# B&R Automation Studio project NAINV104C00R8L515F00 (part 19)

#### Act_Background.st - Do Not Change!!!
```iecst
(** 2022-12-20 **)
ACTION Act_Background:

	pa_tyAlmData[1]	:= tyAlmData;

	IF (bRstErr = TRUE) THEN

		bErr		:= FALSE;
		bWarning	:= FALSE;

		//Reset Warning
		memset(ADR(a_tyWarningCurrList) , 0 , SIZEOF(a_tyWarningCurrList));
		udiWarningMax	:=1;

		memset(ADR(a_tyCurrList) , 0 , SIZEOF(a_tyCurrList));
		memset(ADR(a_sRecoveryList) , 0 , SIZEOF(a_sRecoveryList));
		memset(ADR(a_udiRecoveryList),0,SIZEOF(a_udiRecoveryList));

		udiAlmCntr	:= 0;

		bAlmUpdt	:= FALSE;

	END_IF

	IF (bRstWarning = TRUE) THEN

		IF bErr =FALSE AND bWarning= TRUE THEN
			//Reset Warning
			memset(ADR(a_tyWarningCurrList) , 0 , SIZEOF(a_tyWarningCurrList));
			udiWarningMax	:=1;

			memset(ADR(a_tyCurrList) , 0 , SIZEOF(a_tyCurrList));
			memset(ADR(a_sRecoveryList) , 0 , SIZEOF(a_sRecoveryList));
			memset(ADR(a_udiRecoveryList),0,SIZEOF(a_udiRecoveryList));
			udiAlmCntr	:= 0;
			bWarning := FALSE;
		END_IF

		bAlmUpdt	:= FALSE;

	END_IF

	IF bAlarmLog = TRUE  AND p_bStartupUISettingsLoadDone THEN

		IF (bAlmUpdt = FALSE) OR (eStatus = Error) THEN

			bInfo		:= FALSE;
			bInfoLF		:= FALSE;
			sInfoMsg	:= '';
			iInfoCntr	:= 0;

			FOR udi := 1 TO p_udiCurrMax DO

				IF (pa_tyAlmData[udi].udiRunTime <> a_udiRunTimeOld[udi]) AND pa_tyAlmData[udi].udiCode <> 0
					AND ((pa_tyAlmData[udi].eSeverity = AlmSeverityError ) ) THEN

					a_udiRunTimeOld[udi]	:= pa_tyAlmData[udi].udiRunTime;

					bAlmUpdt	:= TRUE;

					udiAlmCntr	:= udiAlmCntr + 1;
					IF udiAlmCntr > p_udiCurrMax THEN
						udiAlmCntr	:= p_udiCurrMax;
					END_IF

					udiLogCntr	:= udiLogCntr + 1;
					IF udiLogCntr > p_udiCurrMax THEN
						udiLogCntr	:= p_udiCurrMax;
					END_IF

					fLogDTConvert(ADR(sDT) , p_dtCurrDT);
					udiErrorCode := (pa_tyAlmData[udi].udiCode - 10000) + (pa_tyAlmData[udi].udiModuleNum);//*For HMI Text Group*

					//In this case, Program Name/Data Time/
					//Current List
					a_tyCurrList[udiAlmCntr].eSeverity		:= pa_tyAlmData[udi].eSeverity;
					a_tyCurrList[udiAlmCntr].sProgNm		:= pa_tyAlmData[udi].sProgNm;
					a_tyCurrList[udiAlmCntr].sDT			:= sDT;

					//To HMI Text Group
					a_tyCurrList[udiAlmCntr].udiErrorCode	:= udiErrorCode;
					a_tyCurrList[udiAlmCntr].bAlm			:= pa_tyAlmData[udi].bAlm;

					//Recovery List
					a_sRecoveryList[udiAlmCntr]	 			:= pa_tyAlmData[udi].sRcyMsg;
					a_udiRecoveryList[udiAlmCntr]			:= udiErrorCode; //*For HMI Text Group **It will be the same procedure with the above**

					//History List
					memmove(ADR(a_tyHistoryList[2]) , ADR(a_tyHistoryList[1]) , SIZEOF(a_tyHistoryList[1]) * (p_udiHistoryMax - 1));

					a_tyHistoryList[1].sProgNm			:= pa_tyAlmData[udi].sProgNm;
					a_tyHistoryList[1].sDT				:= sDT;
					a_tyHistoryList[1].udiModErrCode	:= pa_tyAlmData[udi].udiCode;
					a_tyHistoryList[1].udiErrorCode		:= udiErrorCode;

					//Log List
					fLogAlmDispMsg(ADR(sAlmMsg) , p_dtCurrDT , pa_tyAlmData[udi].sProgNm , pa_tyAlmData[udi].udiCode , pa_tyAlmData[udi].sAlmMsg); // *For Log files*
					a_sLogList[udiLogCntr]	:= sAlmMsg;
					a_sLogList[udiLogCntr]	:= CONCAT(a_sLogList[udiLogCntr] , '$r$n');

					//Severity
					IF pa_tyAlmData[udi].eSeverity = AlmSeverityError THEN
						bErr		:= TRUE;
					END_IF

					// Alarm warning
				ELSIF (( pa_tyAlmData[udi].eSeverity = AlmSeverityWarning) AND  (pa_tyAlmData[udi].udiCode <> 0 )) THEN

					//Used to compare
					memset(ADR(sWarningCompareMsg) , 0 , SIZEOF(sWarningCompareMsg));

					sWarningCompareMsg	:= CONCAT(sWarningCompareMsg , pa_tyAlmData[udi].sProgNm);
					sWarningCompareMsg	:= CONCAT(sWarningCompareMsg , ' | ');
					sWarningID := UDINT_TO_STRING(pa_tyAlmData[udi].udiCode);
					sWarningCompareMsg	:= CONCAT(sWarningCompareMsg , sWarningID);
					sWarningCompareMsg	:= CONCAT(sWarningCompareMsg , ' | ');
					sWarningCompareMsg	:= CONCAT(sWarningCompareMsg , pa_tyAlmData[udi].sAlmMsg);

					//Checking whether it is recorded in the alarm list
					FOR udi1 := 0 TO  udiWarningMax DO
						WarningListOccur := (memcmp(ADR(sWarningCompareMsg),ADR(a_tyWarningCurrList[udi1].sMsg),SIZEOF(sWarningCompareMsg) )= 0);

						IF WarningListOccur THEN
							EXIT;
						END_IF

					END_FOR

					//IF warning message is no recorded in alarm list
					IF 	WarningListOccur =FALSE THEN

						bAlmUpdt	:= TRUE;
						udiWarningMax := udiWarningMax +1;

						udiAlmCntr	:= udiAlmCntr + 1;

						IF udiAlmCntr > p_udiCurrMax THEN
							udiAlmCntr	:= p_udiCurrMax;
						END_IF

						udiRecorded[udiWarningMax-1]:= udi;

						udiLogCntr	:= udiLogCntr + 1;

						IF udiLogCntr > p_udiCurrMax THEN
							udiLogCntr	:= p_udiCurrMax;
						END_IF

						//Warning List
						a_tyWarningCurrList[udiWarningMax-1].sMsg		:= sWarningCompareMsg;

						fLogDTConvert(ADR(sDT) , p_dtCurrDT);
						udiErrorCode := (pa_tyAlmData[udi].udiCode - 10000) + pa_tyAlmData[udi].udiModuleNum; //*For HMI Text Group*

						//Current List
						a_tyCurrList[udiAlmCntr].eSeverity		:= pa_tyAlmData[udi].eSeverity;
						a_tyCurrList[udiAlmCntr].sProgNm		:= pa_tyAlmData[udi].sProgNm;
						a_tyCurrList[udiAlmCntr].sDT			:= sDT;
						a_tyCurrList[udiAlmCntr].udiModErrCode	:= pa_tyAlmData[udi].udiCode;

						//To HMI Text Group
						a_tyCurrList[udiAlmCntr].udiErrorCode	:= udiErrorCode;
						a_tyCurrList[udiAlmCntr].bWarning		:= pa_tyAlmData[udi].bWarning;

						//Recovery List
						a_sRecoveryList[udiAlmCntr]	 	:= pa_tyAlmData[udi].sRcyMsg;
						a_udiRecoveryList[udiAlmCntr]	:= udiErrorCode;

						//History List
						memmove(ADR(a_tyHistoryList[2]) , ADR(a_tyHistoryList[1]) , SIZEOF(a_tyHistoryList[1]) * (p_udiHistoryMax - 1));

						a_tyHistoryList[1].sProgNm			:= pa_tyAlmData[udi].sProgNm;
						a_tyHistoryList[1].sDT				:= sDT;
						a_tyHistoryList[1].udiModErrCode	:= pa_tyAlmData[udi].udiCode;
						a_tyHistoryList[1].udiErrorCode		:= udiErrorCode;

						//Log List
						//Info Message
						fLogAlmDispMsg(ADR(sWarningMsg) , p_dtCurrDT , pa_tyAlmData[udi].sProgNm , pa_tyAlmData[udi].udiCode , pa_tyAlmData[udi].sAlmMsg);

						a_sLogList[udiLogCntr]	:= sWarningMsg;
						a_sLogList[udiLogCntr]	:= CONCAT(a_sLogList[udiLogCntr] , '$r$n');

						bWarning	:= TRUE;

					END_IF

					// Show Info Message
				ELSIF  ((pa_tyAlmData[udi].udiCode <> 0) AND (pa_tyAlmData[udi].eSeverity = AlmSeverityInfo)) THEN

					iInfoCntr	:= iInfoCntr + 1;

					IF iInfoCntr = 1 THEN
						sInfoMsg	:= pa_tyAlmData[udi].sAlmMsg;

						IF pa_tyAlmData[udi].sProgNm = 'Follower' AND pa_tyAlmData[udi].sAlmMsg <>'' THEN

							bInfoLF	:= TRUE;
							bInfo	:= TRUE;

						ELSE
							bInfoLF	:= FALSE;
							bInfo	:= TRUE;
						END_IF

					ELSIF iInfoCntr = 2 THEN
						sInfoMsg	:= CONCAT(sInfoMsg , '$r$n$r$n');
						sInfoMsg	:= CONCAT(sInfoMsg , pa_tyAlmData[udi].sAlmMsg);

					END_IF

				END_IF

			END_FOR

		ELSE

			p_eAct	:= AlarmActAppendLogWriteHistory;
			IF eStatus = Done AND eStat = AlarmActAppendLogWriteHistory THEN
				p_eAct		:= AlarmActIdle;
				bAlmUpdt	:= FALSE;
				udiLogCntr	:= 0;
			END_IF

		END_IF

	END_IF

END_ACTION
```

#### Act_Alarm.st - Do Not Change!!!
```iecst
(** 2019-03-25 **)
ACTION Act_Alarm:

	//Error
	IF EDGEPOS(eStatus = Error) THEN

		tyAlmData.sProgNm		:= p_sProgNm;
		tyAlmData.udiCode		:= udiStatus;
		tyAlmData.eSeverity		:= AlmSeverityError;
		tyAlmData.udiRunTime	:= tyAlmData.udiRunTime + 1;
		tyAlmData.bAlm			:= TRUE;
		tyAlmData.udiModuleNum  := udiModuleNum;
		g_sAlarmProgNm		:= p_sProgNm;

		//Get Error Message
		IF tyAlmData.udiCode < 10000 OR tyAlmData.udiCode > 10099 THEN
			tyAlmData.sAlmMsg	:= 'Unknown';
			tyAlmData.sRcyMsg	:= 'Unknown';
		ELSE
			tyAlmData.sAlmMsg	:= a_tyAlmText[tyAlmData.udiCode].sAlmText;
			tyAlmData.sRcyMsg	:= a_tyAlmText[tyAlmData.udiCode].sRcyText;
		END_IF

		sStatTxt	:= tyAlmData.sAlmMsg;

	ELSIF bRstErr AND (tyAlmData.udiCode <> 0) THEN

		tyAlmData.udiCode	:= 0;
		tyAlmData.eSeverity	:= AlmSeverityNA;
		tyAlmData.sAlmMsg	:= '';
		tyAlmData.sRcyMsg	:= '';
		tyAlmData.bAlm			:= FALSE;
		sStatTxt	:= a_sStatText[eStat];

	END_IF

END_ACTION
```

#### InputRef.var - Do Not Change!!!
```iecst
(*2022-12-20*)
(**)
(*General*)
VAR
	p_udiCurrMax : REFERENCE TO UDINT;
	p_udiHistoryMax : REFERENCE TO UDINT;
END_VAR
(**)
VAR
	p_eAct : REFERENCE TO eAlarmAction;
	p_udiRstErr : REFERENCE TO UDINT;
END_VAR
(**)
(*Configuration*)
VAR
	p_dtCurrDT : REFERENCE TO DATE_AND_TIME;
	pa_tyAlmData : REFERENCE TO ARRAY[1..c_udiAlarmCurrMax] OF tyAlmDat;
	p_udiFileKeepDay : REFERENCE TO UDINT;
	p_sProgNm : REFERENCE TO STRING[15];
	p_bNtSettingsLoadDone : REFERENCE TO BOOL;
	p_bStartupUISettingsLoadDone : REFERENCE TO BOOL;
END_VAR
```

#### Local.var - Do Not Change!!!
```iecst
(*2022-12-20*)
(**)
(*Local Action, State & Status*)
VAR
	eAct : eAlarmAction := AlarmActIdle;
	eStat : eAlarmAction := AlarmActIdle;
	eStatus : eFBStatus := Idle;
	udiStatus : UDINT := 0;
	sStatTxt : STRING[200] := '';
	a_sStatText : ARRAY[0..50] OF STRING[200] := ['Idling','Creating Directory','Deleting Old Alarm Log File','Reading History File','Writing History File','Appending Alarm Log File','Appending Alarm Log File & Writing History File','Resetting History','Background Start Alarm Log','Background Stop Alarm Log',41('')];
END_VAR
(**)
(*Local Alarm*)
VAR
	tyAlmData : tyAlmDat;
	a_tyAlmText : ARRAY[10000..10099] OF tyAlmTxt := [(sAlmText:='Create User Directory Error',sRcyText:='An Error Occurred While Attempting To Create User Directory. Please Contact Nutek For A Possible Solution'),(sAlmText:='Create Alarm Directory Error',sRcyText:='An Error Occurred While Attempting To Create Alarm Directory. Please Contact Nutek For A Possible Solution'),(sAlmText:='Get Directory Info Error While Deleting Old Log',sRcyText:='An Error Was Encountered While Getting Directory Info. Please Contact Nutek For A Possible Solution.'),(sAlmText:='Directory Read Error While Deleting Old Log',sRcyText:='An Error Was Encountered While Reading Directory. Please Contact Nutek For A Possible Solution.'),(sAlmText:='File Delete Error While Deleting Old Log',sRcyText:='An Error Was Encountered While Trying To Delete File. Please Contact Nutek For A Possible Solution.'),(sAlmText:='File Open Error While Reading Alarm History',sRcyText:='An Error Was Encountered While Trying To Open File. Please Contact Nutek For A Possible Solution.'),(sAlmText:='File Read Error While Reading Alarm History',sRcyText:='An Error Was Encountered While Trying To Read File. Please Contact Nutek For A Possible Solution.'),(sAlmText:='File Close Error While Reading Alarm History',sRcyText:='An Error Was Encountered While Trying To Close File. Please Contact Nutek For A Possible Solution.'),(sAlmText:='File Open Error While Writing Alarm History',sRcyText:='An Error Was Encountered While Trying To Open File. Please Contact Nutek For A Possible Solution.'),(sAlmText:='File Create Error While Writing Alarm History',sRcyText:='An Error Was Encountered While Trying To Create File. Please Contact Nutek For A Possible Solution.'),(sAlmText:='File Write Error While Writing Alarm History',sRcyText:='An Error Was Encountered While Trying To Write File. Please Contact Nutek For A Possible Solution.'),(sAlmText:='File Close Error While Writing Alarm History',sRcyText:='An Error Was Encountered While Trying To Close File. Please Contact Nutek For A Possible Solution.'),(sAlmText:='Directory Does Not Exist While Writing Alarm History',sRcyText:='The Directory Does Not Exist. Please Contact Nutek For A Possible Solution.'),(sAlmText:='File Open Error While Writing Alarm Log',sRcyText:='An Error Was Encountered While Trying To Open File. Please Contact Nutek For A Possible Solution.'),(sAlmText:='File Create Error While Writing Alarm Log',sRcyText:='An Error Was Encountered While Trying To Create File. Please Contact Nutek For A Possible Solution.'),(sAlmText:='Get File Info Error While Writing Alarm Log',sRcyText:='An Error Was Encountered While Getting File Info. Please Contact Nutek For A Possible Solution.'),(sAlmText:='File Write Error While Writing Alarm Log',sRcyText:='An Error Was Encountered While Trying To Write File. Please Contact Nutek For A Possible Solution.'),(sAlmText:='File Close Error While Writing Alarm Log',sRcyText:='An Error Was Encountered While Trying To Close File. Please Contact Nutek For A Possible Solution.'),(sAlmText:='Directory Does Not Exist While Writing Alarm Log',sRcyText:='The Directory Does Not Exist. Please Contact Nutek For A Possible Solution.'),(sAlmText:='File Open Error While Writing Alarm History',sRcyText:='An Error Was Encountered While Trying To Open File. Please Contact Nutek For A Possible Solution.'),(sAlmText:='File Create Error While Writing Alarm History',sRcyText:='An Error Was Encountered While Trying To Create File. Please Contact Nutek For A Possible Solution.'),(sAlmText:='File Write Error While Writing Alarm History',sRcyText:='An Error Was Encountered While Trying To Write File. Please Contact Nutek For A Possible Solution.'),(sAlmText:='File Close Error While Writing Alarm History',sRcyText:='An Error Was Encountered While Trying To Close File. Please Contact Nutek For A Possible Solution.'),(sAlmText:='Directory Does Not Exist While Writing Alarm History',sRcyText:='The Directory Does Not Exist. Please Contact Nutek For A Possible Solution.'),(sAlmText:='File Open Error While Writing Alarm Log',sRcyText:='An Error Was Encountered While Trying To Open File. Please Contact Nutek For A Possible Solution.'),(sAlmText:='File Create Error While Writing Alarm Log',sRcyText:='An Error Was Encountered While Trying To Create File. Please Contact Nutek For A Possible Solution.'),(sAlmText:='Get File Info Error While Writing Alarm Log',sRcyText:='An Error Was Encountered While Getting File Info. Please Contact Nutek For A Possible Solution.'),(sAlmText:='File Write Error While Writing Alarm Log',sRcyText:='An Error Was Encountered While Trying To Write File. Please Contact Nutek For A Possible Solution.'),(sAlmText:='File Close Error While Writing Alarm Log',sRcyText:='An Error Was Encountered While Trying To Close File. Please Contact Nutek For A Possible Solution.'),(sAlmText:='Directory Does Not Exist While Writing Alarm Log',sRcyText:='The Directory Does Not Exist. Please Contact Nutek For A Possible Solution.'),(sAlmText:='File Open Error While Resetting Alarm History',sRcyText:='An Error Was Encountered While Trying To Open File. Please Contact Nutek For A Possible Solution.'),(sAlmText:='File Create Error While Resetting Alarm History',sRcyText:='An Error Was Encountered While Trying To Create File. Please Contact Nutek For A Possible Solution.'),(sAlmText:='File Write Error While Resetting Alarm History',sRcyText:='An Error Was Encountered While Trying To Write File. Please Contact Nutek For A Possible Solution.'),(sAlmText:='File Close Error While Resetting Alarm History',sRcyText:='An Error Was Encountered While Trying To Close File. Please Contact Nutek For A Possible Solution.'),(sAlmText:='Directory Does Not Exist While Resetting Alarm History',sRcyText:='The Directory Does Not Exist. Please Contact Nutek For A Possible Solution.'),65((0))];
END_VAR
(**)
(*Local Output*)
VAR
	bErr : BOOL;
	bWarning : BOOL;
	a_tyCurrList : ARRAY[1..c_udiAlarmCurrMax] OF tyAlarmCurr;
	a_sRecoveryList : ARRAY[1..c_udiAlarmCurrMax] OF STRING[200];
	a_udiRecoveryList : ARRAY[1..c_udiAlarmCurrMax] OF UDINT;
	a_sHistoryList : ARRAY[1..c_udiAlarmHistoryMax] OF STRING[200];
	bInfo : BOOL;
	sInfoMsg : STRING[200];
	bHistoryFileNotFound : BOOL;
	bInfoLF : BOOL := FALSE;
END_VAR
(**)
(*Local Input*)
VAR
	udiRstErr : UDINT := 0;
	dtCurrDT : DATE_AND_TIME;
	a_tyAlmData : ARRAY[1..c_udiAlarmCurrMax] OF tyAlmDat;
	udiFileKeepDay : UDINT := 30;
	sProgNm : STRING[15] := 'Alarm';
	bNtSettingsLoadDone : BOOL := TRUE;
END_VAR
(**)
(*Local*)
VAR
	bRstErr : BOOL;
	udiRstErrOld : UDINT;
	bInitDone : BOOL;
	bInitialDone : BOOL;
	bAlarmLog : BOOL;
	usiStep : USINT;
	udi : UDINT;
	iInfoCntr : INT;
	sAlmMsg : STRING[300];
	udiAlmCntr : UDINT;
	udiAlmRecvryCntr : UDINT;
	udiLogCntr : UDINT;
	udiWriteLogCntr : UDINT;
	a_sLogList : ARRAY[1..c_udiAlarmCurrMax] OF STRING[200];
	bAlmUpdt : BOOL;
	dtCurrDTTemp : DATE_AND_TIME;
	a_udiRunTimeOld : ARRAY[1..c_udiAlarmCurrMax] OF UDINT;
	fbDirCreate1 : fbDirCreate;
	fbDirCreate2 : fbDirCreate;
	fbFileAppend1 : fbFileFullAppend;
	fbFileOldDel1 : fbFileOldDel;
	fbFileRead1 : fbFileFullRead;
	fbFileWrite1 : fbFileFullWrite;
	udi1 : UDINT;
	udi2 : UDINT;
	udiRecorded : ARRAY[1..c_udiAlarmCurrMax] OF UDINT;
	udiRecorded1 : UDINT;
	bRstWarning : BOOL;
	udiWarningMax : UDINT := 1;
	sWarningMsg : STRING[300];
	sWarningID : STRING[80] := '';
	sWarningCompareMsg : STRING[300];
	a_tyWarningCurrList : ARRAY[1..c_udiAlarmCurrMax] OF tyAlarmCurr;
	a_tyHistoryList : ARRAY[1..c_udiAlarmHistoryMax] OF tyHistory;
	WarningListOccur : BOOL := TRUE;
	udiErrorCode : UDINT;
	sDT : STRING[80];
	udiModuleNum : UDINT := 5051;
END_VAR
```

### RstErr.typ - Do Not Change!!!
```iecst
(*2018-12-13*)
(**)
(*Action*)

TYPE
	eRstErrAction :
		(
		RstErrActIdle,
		RstErrActRun,
		RstErrActSetSafetyRlyRst,
		RstErrActRstSafetyRlyRst
		);
END_TYPE
```

### RstErr.var - Change By Project
```iecst
(*2019-03-25*)
(**)
(*Action & State & Status*)
VAR
	p_RstErrStat : UDINT;
	p_RstErrStatus : UDINT;
	p_RstErrStatTxt : UDINT;
END_VAR
(**)
(*Alarm*)
(**)
(*Output*)
VAR
	p_RstErrReset : UDINT;
	p_RstErrSafetyRlyRst : UDINT;
END_VAR
```

### Program Logical/RstErr/RstErr (IEC, version 1.00.0) - 1.00.0 - 

#### Init.st - Change By Project
```iecst
(** 2019-03-25 **)
PROGRAM _INIT

	(* Always Change If Project Change *)

	//Pass Address To Global Address For External Use
	//Action, State & Status
	p_RstErrStat	:= ADR(eStat);
	p_RstErrStatus	:= ADR(eStatus);
	p_RstErrStatTxt	:= ADR(sStatTxt);

	//Alarm

	//Output
	p_RstErrReset			:= ADR(udiRstErr);
	p_RstErrSafetyRlyRst	:= ADR(bSafetyRlyRst);

	(* Always Change If Project Change *)

END_PROGRAM
```

#### Act_InitGlobal.st - Change By Project
```iecst
(** 2019-03-25 **)
ACTION Act_InitGlobal:

	(* Always Change If Project Change *)

	//Pass Data To Link

	//Pass Data To Internal Use
	p_eAct ACCESS p_UIRstErrAct;
	p_bManual ACCESS p_UIUIMnlMod;
	p_bSafetyRlySig ACCESS p_DISafetyRlySig;
	p_bNtSettingsLoadDone ACCESS p_StartupNtSettingsLoadDone;

	(* Always Change If Project Change *)

END_ACTION
```

#### Act_LinkAction.st - Change By Project
```iecst
(** 2019-03-29 **)
ACTION Act_LinkAction:

	IF EDGENEG(p_bManual) THEN
		p_eAct	:= RstErrActIdle;
	END_IF

END_ACTION
```

#### Act_InitLocal.st - Do Not Change!!!
```iecst
(** 2019-03-25 **)
ACTION Act_InitLocal:

	//Input Reference Link To Local Variable
	p_eAct ACCESS ADR(eAct);
	p_bManual ACCESS ADR(bManual);
	p_bSafetyRlySig ACCESS ADR(bSafetyRlySig);
	p_bNtSettingsLoadDone ACCESS ADR(bNtSettingsLoadDone);

END_ACTION
```

#### Act_Initial.st - Do Not Change!!!
```iecst
(** 2019-01-03 **)
ACTION Act_Initial:

	//Initial
	sStatTxt	:= a_sStatText[eStat];

	fbSafetyRlyRstTm(IN := FALSE);

END_ACTION
```

#### Act_Action.st - Do Not Change!!!
```iecst
(** 2019-03-25 **)
ACTION Act_Action:

	//Reset Done
	IF eStatus = Done AND p_eAct = RstErrActIdle THEN
		eStat	:= RstErrActIdle;
	END_IF

	//Set p_eAct
	IF eStatus = Idle THEN
		eStat	:= p_eAct;
	END_IF

END_ACTION
```

#### Act_Main.st - Do Not Change!!!
```iecst
(** 2019-01-18 **)
ACTION Act_Main:

	//Main
	CASE eStat OF

		RstErrActIdle:
			IF eStatus <> Idle THEN	//Reset Data
				//Private
				fbSafetyRlyRstTm(IN := FALSE);

				sStatTxt	:= a_sStatText[eStat];

				IF p_bManual = FALSE THEN
					bSafetyRlyRst	:= FALSE;
				END_IF

			END_IF

			IF EDGENEG(p_bManual) THEN
				bSafetyRlyRst	:= FALSE;
			END_IF

			eStatus	:= Idle;

		RstErrActRun:
			IF eStatus = Idle OR eStatus = Busy THEN

				eStatus	:= Busy;

				sStatTxt	:= a_sStatText[eStat];

				IF bSafetyRlyRst=FALSE THEN
					udiRstErr	:= udiRstErr + 1;
				END_IF

				IF p_bSafetyRlySig = FALSE THEN
					bSafetyRlyRst	:= TRUE;
				END_IF

				IF bSafetyRlyRst = TRUE THEN
					fbSafetyRlyRstTm(IN := TRUE, PT := T#500ms);

					IF fbSafetyRlyRstTm.Q = TRUE THEN
						bSafetyRlyRst	:= FALSE;
						eStatus			:= Done;
					END_IF

				ELSE
					eStatus	:= Done;

				END_IF

			END_IF

		RstErrActSetSafetyRlyRst:
			IF eStatus = Idle OR eStatus = Busy THEN

				sStatTxt	:= a_sStatText[eStat];

				//Reset
				fbSafetyRlyRstTm(IN := FALSE);

				bSafetyRlyRst	:= TRUE;
				eStatus			:= Done;

			END_IF

		RstErrActRstSafetyRlyRst:
			IF eStatus = Idle OR eStatus = Busy THEN

				sStatTxt	:= a_sStatText[eStat];

				//Reset
				fbSafetyRlyRstTm(IN := FALSE);

				bSafetyRlyRst	:= FALSE;
				eStatus			:= Done;

			END_IF

	END_CASE

END_ACTION
```

#### InputRef.var - Do Not Change!!!
```iecst
(*2019-03-25*)
(**)
(*General*)
VAR
	p_eAct : REFERENCE TO eRstErrAction;
END_VAR
(**)
(*Configuration*)
VAR
	p_bManual : REFERENCE TO BOOL;
END_VAR
(**)
(*Input*)
VAR
	p_bSafetyRlySig : REFERENCE TO BOOL;
	p_bNtSettingsLoadDone : REFERENCE TO BOOL;
END_VAR
```

#### Local.var - Do Not Change!!!
```iecst
(*2019-04-30*)
(**)
(*Local Action, State & Status*)
VAR
	eAct : eRstErrAction := RstErrActIdle;
	eStat : eRstErrAction := RstErrActIdle;
	eStatus : eFBStatus := Idle;
	sStatTxt : STRING[200] := '';
	a_sStatText : ARRAY[0..50] OF STRING[200] := ['Idling','Running Reset Error','Turning On Safety Relay Reset','Turning Off Safety Relay Reset',47('')];
END_VAR
(**)
(*Local Alarm*)
(**)
(*Local Output*)
VAR
	udiRstErr : UDINT;
	bSafetyRlyRst : BOOL;
END_VAR
(**)
(*Local Input*)
VAR
	bManual : BOOL := FALSE;
	bSafetyRlySig : BOOL;
	bNtSettingsLoadDone : BOOL := TRUE;
END_VAR
(**)
(*Local*)
VAR
	bInitDone : BOOL;
	bInitialDone : BOOL;
	fbSafetyRlyRstTm : TON;
END_VAR
```

### ProdRcp.typ - Change By Project
```iecst
(*2020-06-08*)
(**)
(*Action*)

TYPE
	eProdRcpAction :
		(
		ProdRcpActIdle,
		ProdRcpActCreateDir,
		ProdRcpActAddEdit,
		ProdRcpActDel,
		ProdRcpActGetInfo,
		ProdRcpActGetList,
		ProdRcpActFilter,
		ProdRcpActLoadRcp,
		ProdRcpActAdd,
		ProdRcpActEdit,
		ProdRcpActReadCurrRcp,
		ProdRcpActWriteCurrRcpParam,
		ProdRcpActSaveList,
		ProdRcpActSort,
		ProdRcpActEndCharFilter
		);
END_TYPE

(**)
(*Data*)

TYPE
	tyProdRcpParam : 	STRUCT
		sRcpNm : STRING[254];
		diWidthInUM : DINT;
		diWidthInUM2 : DINT;
		usiMcMod : USINT;
		sDisplayInfo : STRING[30];
		dtLastModified : DATE_AND_TIME;
		usiFlippedBrd : USINT;
		sMatchCode : STRING[30];
	END_STRUCT;
END_TYPE
```

### ProdRcp.var - Change By Project
```iecst
(*2020-06-08*)
(**)
(*Constant*)
VAR CONSTANT
	c_udiProdRcpMax : UDINT := 2000;
END_VAR
(**)
(*Action & State & Status*)
VAR
	p_ProdRcpStat : UDINT;
	p_ProdRcpStatus : UDINT;
	p_ProdRcpStatTxt : UDINT;
END_VAR
(**)
(*Alarm*)
VAR
	p_ProdRcpAlmData : UDINT;
END_VAR
(**)
(*Output*)
VAR
	p_ProdRcpNmExist : UDINT;
	p_ProdRcpNmNotExist : UDINT;
	p_ProdRcpNmEmpty : UDINT;
	p_ProdRcpListFull : UDINT;
	p_ProdRcpCurrList : UDINT;
	p_ProdRcpFilterList : UDINT;
	p_ProdRcpSortedList : UDINT;
	p_ProdRcpScanList : UDINT;
	p_ProdRcpInfoOut : UDINT;
	p_ProdRcpFileNotFound : UDINT;
	p_ProdRcpCurrRcpAll : UDINT;
END_VAR
(**)
VAR
	p_ProdRcpCurrRcp0 : UDINT;
	p_ProdRcpCurrRcp0Nm : UDINT;
	p_ProdRcpCurrRcp0Width : UDINT;
	p_ProdRcpCurrRcp0McMod : UDINT;
	p_ProdRcpCurrRcp0FlippedBrd : UDINT;
	p_ProdRcpCurrRcp0MatchCode : UDINT;
	p_ProdRcpCurrRcp0DisplayInfo : UDINT;
	p_ProdRcpCurrRcp0LastModified : UDINT;
	p_ProdRcpCurrRcp0Width2 : UDINT;
END_VAR
(**)
VAR
	p_ProdRcpCurrRcp1 : UDINT;
	p_ProdRcpCurrRcp1Nm : UDINT;
	p_ProdRcpCurrRcp1Width : UDINT;
	p_ProdRcpCurrRcp1McMod : UDINT;
	p_ProdRcpCurrRcp1FlippedBrd : UDINT;
	p_ProdRcpCurrRcp1MatchCode : UDINT;
	p_ProdRcpCurrRcp1DisplayInfo : UDINT;
	p_ProdRcpCurrRcp1LastModified : UDINT;
	p_ProdRcpCurrRcp1Width2 : UDINT;
END_VAR
(**)
VAR
	p_ProdRcpCurrRcp2 : UDINT;
	p_ProdRcpCurrRcp2Nm : UDINT;
	p_ProdRcpCurrRcp2Width : UDINT;
	p_ProdRcpCurrRcp2McMod : UDINT;
	p_ProdRcpCurrRcp2FlippedBrd : UDINT;
	p_ProdRcpCurrRcp2MatchCode : UDINT;
	p_ProdRcpCurrRcp2DisplayInfo : UDINT;
	p_ProdRcpCurrRcp2LastModified : UDINT;
	p_ProdRcpCurrRcp2Width2 : UDINT;
END_VAR
(**)
VAR
	p_ProdRcpCurrRcp3 : UDINT;
	p_ProdRcpCurrRcp3Nm : UDINT;
	p_ProdRcpCurrRcp3Width : UDINT;
	p_ProdRcpCurrRcp3McMod : UDINT;
	p_ProdRcpCurrRcp3FlippedBrd : UDINT;
	p_ProdRcpCurrRcp3MatchCode : UDINT;
	p_ProdRcpCurrRcp3DisplayInfo : UDINT;
	p_ProdRcpCurrRcp3LastModified : UDINT;
	p_ProdRcpCurrRcp3Width2 : UDINT;
END_VAR
(**)
VAR
	p_ProdRcpCurrRcp4 : UDINT;
	p_ProdRcpCurrRcp4Nm : UDINT;
	p_ProdRcpCurrRcp4Width : UDINT;
	p_ProdRcpCurrRcp4McMod : UDINT;
	p_ProdRcpCurrRcp4FlippedBrd : UDINT;
	p_ProdRcpCurrRcp4MatchCode : UDINT;
	p_ProdRcpCurrRcp4DisplayInfo : UDINT;
	p_ProdRcpCurrRcp4LastModified : UDINT;
	p_ProdRcpCurrRcp4Width2 : UDINT;
END_VAR
(**)
VAR
	p_ProdRcpCurrRcp5 : UDINT;
	p_ProdRcpCurrRcp5Nm : UDINT;
	p_ProdRcpCurrRcp5Width : UDINT;
	p_ProdRcpCurrRcp5McMod : UDINT;
	p_ProdRcpCurrRcp5FlippedBrd : UDINT;
	p_ProdRcpCurrRcp5MatchCode : UDINT;
	p_ProdRcpCurrRcp5DisplayInfo : UDINT;
	p_ProdRcpCurrRcp5LastModified : UDINT;
	p_ProdRcpCurrRcp5Width2 : UDINT;
END_VAR
```

### Program Logical/ProdRcp/ProdRcp (IEC, version 1.00.0) - 1.00.0 - NtRecipe v5.00.0 , NtFileIO v5.00.0 (2018-12-01)

#### Init.st - Change By Project
```iecst
(** 2019-06-10 **)
PROGRAM _INIT

	(* Always Change If Project Change *)

	//Pass Address To Global Address For External Use
	//Action, State & Status
	p_ProdRcpStat		:= ADR(eStat);
	p_ProdRcpStatus		:= ADR(eStatus);
	p_ProdRcpStatTxt	:= ADR(sStatTxt);

	//Alarm
	p_ProdRcpAlmData	:= ADR(tyAlmData);

	//Output
	p_ProdRcpNmExist				:= ADR(bNmExist);
	p_ProdRcpNmNotExist				:= ADR(bNmNotExist);
	p_ProdRcpNmEmpty				:= ADR(bNmEmpty);
	p_ProdRcpListFull				:= ADR(bListFull);
	p_ProdRcpCurrList				:= ADR(a_tyCurrList);
	p_ProdRcpFilterList				:= ADR(a_tyFilterList);
	p_ProdRcpSortedList				:= ADR(a_tySortList);
	p_ProdRcpScanList				:= ADR(a_tyScanList);
	p_ProdRcpInfoOut				:= ADR(tyInfoOut);
	p_ProdRcpFileNotFound			:= ADR(bFileNotFound);
	p_ProdRcpCurrRcpAll				:= ADR(a_tyCurrRcp);
	p_ProdRcpCurrRcp0				:= ADR(a_tyCurrRcp[0]);
	p_ProdRcpCurrRcp0Nm				:= ADR(a_tyCurrRcp[0].sRcpNm);
	p_ProdRcpCurrRcp0Width			:= ADR(a_tyCurrRcp[0].diWidthInUM);
	p_ProdRcpCurrRcp0McMod			:= ADR(a_tyCurrRcp[0].usiMcMod);
	p_ProdRcpCurrRcp0FlippedBrd		:= ADR(a_tyCurrRcp[0].usiFlippedBrd);
	p_ProdRcpCurrRcp0MatchCode		:= ADR(a_tyCurrRcp[0].sMatchCode);
	p_ProdRcpCurrRcp0DisplayInfo	:= ADR(a_tyCurrRcp[0].sDisplayInfo);
	p_ProdRcpCurrRcp0LastModified	:= ADR(a_tyCurrRcp[0].dtLastModified);
	p_ProdRcpCurrRcp0Width2			:= ADR(a_tyCurrRcp[0].diWidthInUM2);

	p_ProdRcpCurrRcp1				:= ADR(a_tyCurrRcp[1]);
	p_ProdRcpCurrRcp1Nm				:= ADR(a_tyCurrRcp[1].sRcpNm);
	p_ProdRcpCurrRcp1Width			:= ADR(a_tyCurrRcp[1].diWidthInUM);
	p_ProdRcpCurrRcp1McMod			:= ADR(a_tyCurrRcp[1].usiMcMod);
	p_ProdRcpCurrRcp1FlippedBrd		:= ADR(a_tyCurrRcp[1].usiFlippedBrd);
	p_ProdRcpCurrRcp1MatchCode		:= ADR(a_tyCurrRcp[1].sMatchCode);
	p_ProdRcpCurrRcp1DisplayInfo	:= ADR(a_tyCurrRcp[1].sDisplayInfo);
	p_ProdRcpCurrRcp1LastModified	:= ADR(a_tyCurrRcp[1].dtLastModified);
	p_ProdRcpCurrRcp1Width2			:= ADR(a_tyCurrRcp[1].diWidthInUM2);

	p_ProdRcpCurrRcp2				:= ADR(a_tyCurrRcp[2]);
	p_ProdRcpCurrRcp2Nm				:= ADR(a_tyCurrRcp[2].sRcpNm);
	p_ProdRcpCurrRcp2Width			:= ADR(a_tyCurrRcp[2].diWidthInUM);
	p_ProdRcpCurrRcp2McMod			:= ADR(a_tyCurrRcp[2].usiMcMod);
	p_ProdRcpCurrRcp2FlippedBrd		:= ADR(a_tyCurrRcp[2].usiFlippedBrd);
	p_ProdRcpCurrRcp2MatchCode		:= ADR(a_tyCurrRcp[2].sMatchCode);
	p_ProdRcpCurrRcp2DisplayInfo	:= ADR(a_tyCurrRcp[2].sDisplayInfo);
	p_ProdRcpCurrRcp2LastModified	:= ADR(a_tyCurrRcp[2].dtLastModified);
	p_ProdRcpCurrRcp2Width2			:= ADR(a_tyCurrRcp[2].diWidthInUM2);

	p_ProdRcpCurrRcp3				:= ADR(a_tyCurrRcp[3]);
	p_ProdRcpCurrRcp3Nm				:= ADR(a_tyCurrRcp[3].sRcpNm);
	p_ProdRcpCurrRcp3Width			:= ADR(a_tyCurrRcp[3].diWidthInUM);
	p_ProdRcpCurrRcp3McMod			:= ADR(a_tyCurrRcp[3].usiMcMod);
	p_ProdRcpCurrRcp3FlippedBrd		:= ADR(a_tyCurrRcp[3].usiFlippedBrd);
	p_ProdRcpCurrRcp3MatchCode		:= ADR(a_tyCurrRcp[3].sMatchCode);
	p_ProdRcpCurrRcp3DisplayInfo	:= ADR(a_tyCurrRcp[3].sDisplayInfo);
	p_ProdRcpCurrRcp3LastModified	:= ADR(a_tyCurrRcp[3].dtLastModified);
	p_ProdRcpCurrRcp3Width2			:= ADR(a_tyCurrRcp[3].diWidthInUM2);

	p_ProdRcpCurrRcp4				:= ADR(a_tyCurrRcp[4]);
	p_ProdRcpCurrRcp4Nm				:= ADR(a_tyCurrRcp[4].sRcpNm);
	p_ProdRcpCurrRcp4Width			:= ADR(a_tyCurrRcp[4].diWidthInUM);
	p_ProdRcpCurrRcp4McMod			:= ADR(a_tyCurrRcp[4].usiMcMod);
	p_ProdRcpCurrRcp4FlippedBrd		:= ADR(a_tyCurrRcp[4].usiFlippedBrd);
	p_ProdRcpCurrRcp4MatchCode		:= ADR(a_tyCurrRcp[4].sMatchCode);
	p_ProdRcpCurrRcp4DisplayInfo	:= ADR(a_tyCurrRcp[4].sDisplayInfo);
	p_ProdRcpCurrRcp4LastModified	:= ADR(a_tyCurrRcp[4].dtLastModified);
	p_ProdRcpCurrRcp4Width2			:= ADR(a_tyCurrRcp[4].diWidthInUM2);

	p_ProdRcpCurrRcp5				:= ADR(a_tyCurrRcp[5]);
	p_ProdRcpCurrRcp5Nm				:= ADR(a_tyCurrRcp[5].sRcpNm);
	p_ProdRcpCurrRcp5Width			:= ADR(a_tyCurrRcp[5].diWidthInUM);
	p_ProdRcpCurrRcp5McMod			:= ADR(a_tyCurrRcp[5].usiMcMod);
	p_ProdRcpCurrRcp5FlippedBrd		:= ADR(a_tyCurrRcp[5].usiFlippedBrd);
	p_ProdRcpCurrRcp5MatchCode		:= ADR(a_tyCurrRcp[5].sMatchCode);
	p_ProdRcpCurrRcp5DisplayInfo	:= ADR(a_tyCurrRcp[5].sDisplayInfo);
	p_ProdRcpCurrRcp5LastModified	:= ADR(a_tyCurrRcp[5].dtLastModified);
	p_ProdRcpCurrRcp5Width2			:= ADR(a_tyCurrRcp[5].diWidthInUM2);

	(* Always Change If Project Change *)

END_PROGRAM
```

#### Act_InitGlobal.st - Change By Project
```iecst
(** 2020-06-08 **)
ACTION Act_InitGlobal:

	(* Always Change If Project Change *)

	//Pass Data To Link
	p_bLinkStartupRun ACCESS p_StartupRun;
	p_bLinkNtParamLCSManageRcpPrep ACCESS p_NtParamLCSManageRcpPrep;
	p_bLinkMcParamLCSManageRcpEn ACCESS p_McParamLCSManageRcpEn;
	p_eLinkLCSMngRcpProdRcpAct ACCESS p_LCSMngRcpProdRcpAct;
	p_eLinkUIProdRcpAct ACCESS p_UIProdRcpAct;

	//Pass Data To Internal Use
	p_udiRstErr ACCESS p_RstErrReset;
	p_dtCurrDT ACCESS p_TimeCurrDT;
	p_sSearch ACCESS p_UIProdRcpSearch;
	p_sScan ACCESS p_UIProdRcpScan;
	p_tyInfoIn ACCESS p_UIProdRcpInfoIn;
	p_tyCurrRcpWr ACCESS p_UIProdRcpCurrRcpWr;
	p_sListFileName ACCESS p_NtParamProdRcpListFileNm;
	p_sSingleFileName ACCESS p_NtParamProdRcpSingleFileNm;
	p_sProgNm ACCESS p_NtParamProdRcpProgNm;
	p_bNtSettingsLoadDone ACCESS p_StartupNtSettingsLoadDone;

	p_bWidth2Prep ACCESS p_NtParamLFWidth2Prep;
	(* Always Change If Project Change *)

END_ACTION
```

#### InputRef_Link.var - Change By Project
```iecst
(*2019-04-24*)
(**)
VAR
	rWidthInMM : REAL;
	rWidthInMM2 : REAL;
	sWidthInMM : STRING[30];
	sWidthInMM2 : STRING[30];
	p_bLinkStartupRun : REFERENCE TO BOOL;
	p_bLinkNtParamLCSManageRcpPrep : REFERENCE TO BOOL;
	p_bLinkMcParamLCSManageRcpEn : REFERENCE TO BOOL;
	p_eLinkLCSMngRcpProdRcpAct : REFERENCE TO eProdRcpAction;
	p_eLinkUIProdRcpAct : REFERENCE TO eProdRcpAction;
	udi : UDINT;
	udiSortCurrenTotalCntr : UDINT;
	iSortCurrentOuterCntr : INT;
	iTotalRcp : INT;
	iSortCurrentInnerCntr : INT;
	sDebug : STRING[300];
	tyTempRecipe : tyProdRcpParam;
END_VAR
```

#### Act_LinkAction.st - Change By Project
```iecst
(** 2019-05-20 **)
ACTION Act_LinkAction:

	IF p_bLinkStartupRun = TRUE THEN
		p_eAct ACCESS p_StartupProdRcpAct;
	ELSE
		IF eStatus = Idle THEN
			IF p_bLinkNtParamLCSManageRcpPrep AND p_bLinkMcParamLCSManageRcpEn THEN
				IF p_eLinkLCSMngRcpProdRcpAct <> ProdRcpActIdle THEN
					p_eAct ACCESS p_LCSMngRcpProdRcpAct;
					p_tyInfoIn ACCESS p_LCSMngRcpProdRcpInfoIn;
				ELSIF p_eLinkUIProdRcpAct <> ProdRcpActIdle THEN
					p_eAct ACCESS p_UIProdRcpAct;
					p_tyInfoIn ACCESS p_UIProdRcpInfoIn;

					p_tyInfoIn.dtLastModified	:= p_dtCurrDT;
				END_IF
			ELSE
				p_eAct ACCESS p_UIProdRcpAct;
				p_tyInfoIn ACCESS p_UIProdRcpInfoIn;

				p_tyInfoIn.dtLastModified	:= p_dtCurrDT;
			END_IF
		END_IF
	END_IF

END_ACTION
```

#### Act_Link.st - Change By Project
```iecst
(** 2019-04-30 **)
ACTION Act_Link:

	IF (p_eAct = ProdRcpActAddEdit) OR (p_eAct = ProdRcpActAdd) OR (p_eAct = ProdRcpActEdit) THEN

		rWidthInMM				:= DINT_TO_REAL(p_tyInfoIn.diWidthInUM);
		rWidthInMM2				:= DINT_TO_REAL(p_tyInfoIn.diWidthInUM2);
		rWidthInMM				:= rWidthInMM / 1000;
		rWidthInMM2				:= rWidthInMM2 / 1000;
		sWidthInMM				:= REAL_TO_STRING(rWidthInMM);
		sWidthInMM2				:= REAL_TO_STRING(rWidthInMM2);

		IF p_bWidth2Prep THEN
			p_tyInfoIn.sDisplayInfo	:= sWidthInMM;
			p_tyInfoIn.sDisplayInfo	:= CONCAT(p_tyInfoIn.sDisplayInfo , ' | ');
			p_tyInfoIn.sDisplayInfo	:= CONCAT(p_tyInfoIn.sDisplayInfo , sWidthInMM2);
			p_tyInfoIn.sDisplayInfo	:= CONCAT(p_tyInfoIn.sDisplayInfo , ' mm');
		ELSE
			p_tyInfoIn.sDisplayInfo	:= sWidthInMM;
			p_tyInfoIn.sDisplayInfo	:= CONCAT(p_tyInfoIn.sDisplayInfo , ' mm');
		END_IF
	END_IF

END_ACTION
```

#### Cyclic.st - Do Not Change!!!
```iecst
(** 2019-03-29 **)
PROGRAM _CYCLIC

	IF bInitDone = FALSE THEN
		bInitDone	:= TRUE;

		Act_InitLocal;
		Act_InitGlobal;

	ELSIF bInitialDone = FALSE THEN
		IF p_bNtSettingsLoadDone = TRUE THEN
			bInitialDone	:= TRUE;

			Act_Initial;
		END_IF

	ELSE

		Act_RstErr;
		Act_LinkAction;
		Act_Action;
		Act_Link;
		Act_Main;
		Act_Alarm;

	END_IF

END_PROGRAM
```

#### Act_InitLocal.st - Do Not Change!!!
```iecst
(** 2020-06-08 **)
ACTION Act_InitLocal:

	//Input Reference Link To Local Variable
	p_eAct ACCESS ADR(eAct);
	p_udiMax ACCESS ADR(c_udiProdRcpMax);
	p_udiRstErr ACCESS ADR(udiRstErr);
	p_dtCurrDT ACCESS ADR(dtCurrDT);
	p_sSearch ACCESS ADR(sSearch);
	p_sScan ACCESS ADR(sScan);
	p_tyInfoIn ACCESS ADR(tyInfoIn);
	p_tyCurrRcpWr ACCESS ADR(tyCurrRcpWr);
	p_sListFileName ACCESS ADR(sListFileName);
	p_sSingleFileName ACCESS ADR(sSingleFileName);
	p_sProgNm ACCESS ADR(sProgNm);
	p_bNtSettingsLoadDone ACCESS ADR(bNtSettingsLoadDone);
	p_bWidth2Prep ACCESS ADR(bWidth2Prep);

END_ACTION
```

#### Act_Initial.st - Do Not Change!!!
```iecst
(** 2019-06-10 **)
ACTION Act_Initial:

	//Initial
	sStatTxt	:= a_sStatText[eStat];

	fbDirCreate1.sDevice	:= 'F';
	fbDirCreate1.sDirName	:= 'User';
	fbDirCreate1(bEn := FALSE);

	fbDirCreate2.sDevice	:= 'User';
	fbDirCreate2.sDirName	:= 'ProductRecipe';
	fbDirCreate2(bEn := FALSE);

	fbFileReadList.sDevice		:= 'ProdRcp';
	fbFileReadList.sFile		:= p_sListFileName;
	fbFileReadList.udiOffset	:= 0;
	fbFileReadList.p_Dest		:= ADR(a_tyCurrList);
	fbFileReadList.udiLen		:= SIZEOF(a_tyCurrList);
	fbFileReadList(bEn := FALSE);

	fbFileWriteList.sDevice		:= 'ProdRcp';
	fbFileWriteList.sFile		:= p_sListFileName;
	fbFileWriteList.udiOffset	:= 0;
	fbFileWriteList.p_Src		:= ADR(a_tyListTemp);
	fbFileWriteList.udiLen		:= SIZEOF(a_tyListTemp);
	fbFileWriteList.udiOption	:= 0;
	fbFileWriteList(bEn := FALSE);

	fbFileReadSingle.sDevice	:= 'ProdRcp';
	fbFileReadSingle.sFile		:= p_sSingleFileName;
	fbFileReadSingle.udiOffset	:= 0;
	fbFileReadSingle.p_Dest		:= ADR(a_tyCurrRcp[0]);
	fbFileReadSingle.udiLen		:= SIZEOF(a_tyCurrRcp[0]);
	fbFileReadSingle(bEn := FALSE);

	fbFileLoadSingle.sDevice	:= 'ProdRcp';
	fbFileLoadSingle.sFile		:= p_sSingleFileName;
	fbFileLoadSingle.udiOffset	:= 0;
	fbFileLoadSingle.p_Src		:= ADR(a_tyCurrRcp[0]);
	fbFileLoadSingle.udiLen		:= SIZEOF(a_tyCurrRcp[0]);
	fbFileLoadSingle.udiOption	:= 0;
	fbFileLoadSingle(bEn := FALSE);

	fbFileWriteSingle.sDevice	:= 'ProdRcp';
	fbFileWriteSingle.sFile		:= p_sSingleFileName;
	fbFileWriteSingle.udiOffset	:= 0;
	fbFileWriteSingle.p_Src		:= ADR(p_tyCurrRcpWr);
	fbFileWriteSingle.udiLen	:= SIZEOF(p_tyCurrRcpWr);
	fbFileWriteSingle.udiOption	:= 0;
	fbFileWriteSingle(bEn := FALSE);

END_ACTION
```

#### Act_Action.st - Do Not Change!!!
```iecst
(** 2019-03-25 **)
ACTION Act_Action:

	//Reset Error
	IF (eStatus = Error) AND bRstErr THEN
		p_eAct	:= ProdRcpActIdle;
		eStat	:= ProdRcpActIdle;
	END_IF

	//Reset Done
	IF eStatus = Done AND p_eAct = ProdRcpActIdle THEN
		eStat	:= ProdRcpActIdle;
	END_IF

	//Set p_eAct
	IF eStatus = Idle THEN
		eStat	:= p_eAct;
	END_IF

END_ACTION
```

#### Act_Main.st - Do Not Change!!!
```iecst
(** 2023-02-13 **)
ACTION Act_Main:

	//Main
	CASE eStat OF

		ProdRcpActIdle:
			IF eStatus <> Idle THEN	//Reset Data
				//Private
				fbDirCreate1(bEn := FALSE);
				fbDirCreate2(bEn := FALSE);
				fbFileReadList(bEn := FALSE);
				fbFileWriteList(bEn := FALSE);
				fbFileReadSingle(bEn := FALSE);
				fbFileWriteSingle(bEn := FALSE);
				fbFileLoadSingle(bEn := FALSE);
				usiStep				:= 0;
				udiAddStatus		:= 0;

				bNmExist		:= FALSE;
				bNmNotExist		:= FALSE;
				bNmEmpty		:= FALSE;
				bListFull		:= FALSE;
				bFileNotFound	:= FALSE;
				iTotalRcp 		:= 0;

				memset(ADR(tyTempRecipe), 0 , SIZEOF(tyTempRecipe));

				sStatTxt	:= a_sStatText[eStat];

			END_IF

			eStatus	:= Idle;

		ProdRcpActCreateDir:
			IF eStatus = Idle OR eStatus = Busy THEN

				eStatus	:= Busy;

				sStatTxt	:= a_sStatText[eStat];

				CASE usiStep OF
					0:
						fbDirCreate1(bEn := TRUE);
						IF fbDirCreate1.udiStatus = 0 THEN
							usiStep	:= 1;
						ELSIF fbDirCreate1.udiStatus < 65534 THEN
							eStatus		:= Error;

							IF fbDirCreate1.udiStatus = 1908 THEN
								udiStatus	:= 10000;	//Create User Directory Error
							ELSE
								udiStatus	:= fbDirCreate1.udiStatus;
							END_IF
						END_IF

					1:
						fbDirCreate2(bEn := TRUE);
						IF fbDirCreate2.udiStatus = 0 THEN
							eStatus	:= Done;
						ELSIF fbDirCreate2.udiStatus < 65534 THEN
							eStatus		:= Error;

							IF fbDirCreate2.udiStatus = 1908 THEN
								udiStatus	:= 10001;	//Create Product Recipe Directory Error
							ELSE
								udiStatus	:= fbDirCreate2.udiStatus;
							END_IF
						END_IF

				END_CASE

			END_IF

		ProdRcpActAddEdit:
			IF eStatus = Idle OR eStatus = Busy THEN

				eStatus	:= Busy;

				sStatTxt	:= a_sStatText[eStat];

				CASE usiStep OF
					0:	//Edit Recipe
						udiAddStatus	:= fRecipeAddEdit(ADR(p_tyInfoIn) , ADR(a_tyListTemp) , SIZEOF(a_tyListTemp[1]) , ADR(a_tyListTemp[1].sRcpNm) , SIZEOF(a_tyListTemp[1].sRcpNm) , p_udiMax);

						IF udiAddStatus = 1600 THEN	//Recipe Name Empty
							bNmEmpty	:= TRUE;
							eStatus		:= Done;

						ELSIF udiAddStatus = 1601 THEN	//Recipe Full
							bListFull	:= TRUE;
							eStatus		:= Done;

						ELSIF udiAddStatus = 0 THEN	//OK
							usiStep	:= 1;

						END_IF

					1:	//Write Into File
						fbFileWriteList(bEn := TRUE);

						IF fbFileWriteList.udiStatus = 0 THEN
							a_tyCurrList	:= a_tyListTemp;

							eStatus := Done;

						ELSIF fbFileWriteList.udiStatus < 65534 THEN
							a_tyListTemp	:= a_tyCurrList;
							eStatus			:= Error;

							IF fbFileWriteList.udiStatus = 1900 THEN
								udiStatus	:= 10002;	//File Open Error While Adding & Editing
							ELSIF fbFileWriteList.udiStatus = 1901 THEN
								udiStatus	:= 10003;	//File Create Error While Adding & Editing
							ELSIF fbFileWriteList.udiStatus = 1903 THEN
								udiStatus	:= 10004;	//File Write Error While Adding & Editing
							ELSIF fbFileWriteList.udiStatus = 1904 THEN
								udiStatus	:= 10005;	//File Close Error While Adding & Editing
							ELSIF fbFileWriteList.udiStatus = 1914 THEN
								udiStatus	:= 10013;	//Directory Does Not Exist While Adding & Editing
							ELSE
								udiStatus	:= fbFileWriteList.udiStatus;
							END_IF
						END_IF

				END_CASE

			END_IF

		ProdRcpActDel:
			IF eStatus = Idle OR eStatus = Busy THEN

				eStatus	:= Busy;

				sStatTxt	:= a_sStatText[eStat];

				CASE usiStep OF
					0:	//Edit User
						udiAddStatus	:= fRecipeDelete(ADR(p_tyInfoIn) , ADR(a_tyListTemp) , SIZEOF(a_tyListTemp[1]) , ADR(a_tyListTemp[1].sRcpNm) , SIZEOF(a_tyListTemp[1].sRcpNm) , p_udiMax);

						IF udiAddStatus = 1600 THEN	//Recipe Name Empty
							bNmEmpty	:= TRUE;
							eStatus		:= Done;

						ELSIF udiAddStatus = 1603 THEN	//Recipe Not Exist
							bNmNotExist	:= TRUE;
							eStatus		:= Done;

						ELSIF udiAddStatus = 0 THEN	//OK
							usiStep	:= 1;

						END_IF

					1:	//Write Into File
						fbFileWriteList(bEn := TRUE);

						IF fbFileWriteList.udiStatus = 0 THEN
							a_tyCurrList	:= a_tyListTemp;
							eStatus := Done;

						ELSIF fbFileWriteList.udiStatus < 65534 THEN
							a_tyListTemp	:= a_tyCurrList;
							eStatus			:= Error;

							IF fbFileWriteList.udiStatus = 1900 THEN
								udiStatus	:= 10006;	//File Open Error While Deleting
							ELSIF fbFileWriteList.udiStatus = 1901 THEN
								udiStatus	:= 10007;	//File Create Error While Deleting
							ELSIF fbFileWriteList.udiStatus = 1903 THEN
								udiStatus	:= 10008;	//File Write Error While Deleting
							ELSIF fbFileWriteList.udiStatus = 1904 THEN
								udiStatus	:= 10009;	//File Close Error While Deleting
							ELSIF fbFileWriteList.udiStatus = 1914 THEN
								udiStatus	:= 10014;	//Directory Does Not Exist While Deleting
							ELSE
								udiStatus	:= fbFileWriteList.udiStatus;
							END_IF

						END_IF

				END_CASE

			END_IF

		ProdRcpActGetInfo:
			IF eStatus = Idle OR eStatus = Busy THEN

				sStatTxt	:= a_sStatText[eStat];

				IF p_tyInfoIn.sRcpNm = '' THEN
					bNmEmpty	:= TRUE;
					bNmNotExist	:= TRUE;
				ELSE
					bNmNotExist	:= (fRecipeGetInfo(p_tyInfoIn.sRcpNm , ADR(tyInfoOut) , ADR(a_tyCurrList) , SIZEOF(a_tyCurrList[1]) , ADR(a_tyCurrList[1].sRcpNm) , SIZEOF(a_tyCurrList[1].sRcpNm) , p_udiMax)) = 0;
				END_IF

				eStatus	:= Done;

			END_IF

		ProdRcpActGetList:
			IF eStatus = Idle OR eStatus = Busy THEN

				eStatus	:= Busy;

				sStatTxt	:= a_sStatText[eStat];

				fbFileReadList(bEn := TRUE);

				IF fbFileReadList.udiStatus = 0 THEN
					a_tyListTemp	:= a_tyCurrList;
					eStatus			:= Done;

				ELSIF fbFileReadList.udiStatus < 65534 THEN
					eStatus		:= Error;

					IF fbFileReadList.udiStatus = 1900 THEN
						udiStatus	:= 10010;	//File Open Error While Getting List
					ELSIF fbFileReadList.udiStatus = 1902 THEN
						udiStatus	:= 10011;	//File Read Error While Getting List
					ELSIF fbFileReadList.udiStatus = 1904 THEN
						udiStatus	:= 10012;	//File Close Error While Getting List
					ELSIF fbFileReadList.udiStatus = 1915 THEN
						eStatus			:= Done;
						bFileNotFound	:= TRUE;
					ELSE
						udiStatus	:= fbFileReadList.udiStatus;
					END_IF

				END_IF

			END_IF

		ProdRcpActFilter:

			IF eStatus = Idle OR eStatus = Busy THEN

				eStatus := Busy;

				sStatTxt	:= a_sStatText[eStat];

				CASE usiStep OF
					0:
						fRecipeFilter(p_sSearch , ADR(a_tyFilterList) , ADR(a_tyCurrList) , SIZEOF(a_tyCurrList[1]) , ADR(a_tyCurrList[1].sRcpNm) ,
						SIZEOF(a_tyCurrList[1].sRcpNm) , p_udiMax, 0, 499, iFilterCtr);
						usiStep := 1;
					1:
						fRecipeFilter(p_sSearch , ADR(a_tyFilterList) , ADR(a_tyCurrList) , SIZEOF(a_tyCurrList[1]) , ADR(a_tyCurrList[1].sRcpNm) ,
						SIZEOF(a_tyCurrList[1].sRcpNm) , p_udiMax, 500, 999, iFilterCtr);
						usiStep := 2;
					2:
						fRecipeFilter(p_sSearch , ADR(a_tyFilterList) , ADR(a_tyCurrList) , SIZEOF(a_tyCurrList[1]) , ADR(a_tyCurrList[1].sRcpNm) ,
						SIZEOF(a_tyCurrList[1].sRcpNm) , p_udiMax, 1000, 1499, iFilterCtr);
						usiStep := 3;
					3:
						fRecipeFilter(p_sSearch , ADR(a_tyFilterList) , ADR(a_tyCurrList) , SIZEOF(a_tyCurrList[1]) , ADR(a_tyCurrList[1].sRcpNm) ,
						SIZEOF(a_tyCurrList[1].sRcpNm) , p_udiMax, 1500, 1999, iFilterCtr);
						eStatus := Done;

				END_CASE

			END_IF

		ProdRcpActLoadRcp:
			IF eStatus = Idle OR eStatus = Busy THEN

				sStatTxt	:= a_sStatText[eStat];

				CASE usiStep OF
					0:	//Get Current Recipe
						IF p_tyInfoIn.sRcpNm = '' THEN
							bNmEmpty	:= TRUE;
							bNmNotExist	:= TRUE;

							eStatus	:= Done;
						ELSE
							bNmNotExist	:= (fRecipeGetInfo(p_tyInfoIn.sRcpNm , ADR(a_tyCurrRcp[0]) , ADR(a_tyCurrList) , SIZEOF(a_tyCurrList[1]) , ADR(a_tyCurrList[1].sRcpNm) , SIZEOF(a_tyCurrList[1].sRcpNm) , p_udiMax)) = 0;

							IF bNmNotExist = TRUE THEN
								eStatus	:= Done;
							ELSE
								usiStep	:= 1;
							END_IF

						END_IF

					1:	//Write Into File
						fbFileLoadSingle(bEn := TRUE);

						IF fbFileLoadSingle.udiStatus = 0 THEN
							eStatus			:= Done;
						ELSIF fbFileLoadSingle.udiStatus < 65534 THEN
							eStatus			:= Error;

							IF fbFileLoadSingle.udiStatus = 1900 THEN
								udiStatus	:= 10025;	//File Open Error While Loading Current Recipe
							ELSIF fbFileLoadSingle.udiStatus = 1901 THEN
								udiStatus	:= 10026;	//File Create Error While Loading Current Recipe
							ELSIF fbFileLoadSingle.udiStatus = 1903 THEN
								udiStatus	:= 10027;	//File Write Error While Loading Current Recipe
							ELSIF fbFileLoadSingle.udiStatus = 1904 THEN
								udiStatus	:= 10028;	//File Close Error While Loading Current Recipe
							ELSIF fbFileLoadSingle.udiStatus = 1914 THEN
								udiStatus	:= 10029;	//Directory Does Not Exist While Loading Current Recipe
							ELSE
								udiStatus	:= fbFileLoadSingle.udiStatus;
							END_IF
						END_IF

				END_CASE

			END_IF

		ProdRcpActAdd:
			IF eStatus = Idle OR eStatus = Busy THEN

				eStatus	:= Busy;

				sStatTxt	:= a_sStatText[eStat];

				CASE usiStep OF
					0:	//Edit Recipe
						udiAddStatus	:= fRecipeAdd(ADR(p_tyInfoIn) , ADR(a_tyListTemp) , SIZEOF(a_tyListTemp[1]) , ADR(a_tyListTemp[1].sRcpNm) , SIZEOF(a_tyListTemp[1].sRcpNm) , p_udiMax);

						IF udiAddStatus = 1600 THEN	//Recipe Name Empty
							bNmEmpty	:= TRUE;
							eStatus		:= Done;

						ELSIF udiAddStatus = 1601 THEN	//Recipe Full
							bListFull	:= TRUE;
							eStatus		:= Done;

						ELSIF udiAddStatus = 1602 THEN	//Recipe Name Exist
							bNmExist	:= TRUE;
							eStatus		:= Done;

						ELSIF udiAddStatus = 0 THEN	//OK
							usiStep	:= 1;

						END_IF

					1:	//Write Into File
						fbFileWriteList(bEn := TRUE);

						IF fbFileWriteList.udiStatus = 0 THEN
							a_tyCurrList	:= a_tyListTemp;
							eStatus			:= Done;

						ELSIF fbFileWriteList.udiStatus < 65534 THEN
							a_tyListTemp	:= a_tyCurrList;
							eStatus			:= Error;

							IF fbFileWriteList.udiStatus = 1900 THEN
								udiStatus	:= 10015;	//File Open Error While Adding
							ELSIF fbFileWriteList.udiStatus = 1901 THEN
								udiStatus	:= 10016;	//File Create Error While Adding
							ELSIF fbFileWriteList.udiStatus = 1903 THEN
								udiStatus	:= 10017;	//File Write Error While Adding
							ELSIF fbFileWriteList.udiStatus = 1904 THEN
								udiStatus	:= 10018;	//File Close Error While Adding
							ELSIF fbFileWriteList.udiStatus = 1914 THEN
								udiStatus	:= 10019;	//Directory Does Not Exist While Adding
							ELSE
								udiStatus	:= fbFileWriteList.udiStatus;
							END_IF
						END_IF
				END_CASE

			END_IF

		ProdRcpActEdit:
			IF eStatus = Idle OR eStatus = Busy THEN

				eStatus	:= Busy;

				sStatTxt	:= a_sStatText[eStat];

				CASE usiStep OF
					0:	//Edit Recipe
						udiAddStatus	:= fRecipeEdit(ADR(p_tyInfoIn) , ADR(a_tyListTemp) , SIZEOF(a_tyListTemp[1]) , ADR(a_tyListTemp[1].sRcpNm) , SIZEOF(a_tyListTemp[1].sRcpNm) , p_udiMax);

						IF udiAddStatus = 1600 THEN	//Recipe Name Empty
							bNmEmpty	:= TRUE;
							eStatus		:= Done;

						ELSIF udiAddStatus = 1603 THEN	//Recipe Not Exist
							bNmNotExist	:= TRUE;
							eStatus		:= Done;

						ELSIF udiAddStatus = 0 THEN	//OK
							usiStep	:= 1;

						END_IF

					1:	//Write Into File
						fbFileWriteList(bEn := TRUE);

						IF fbFileWriteList.udiStatus = 0 THEN
							a_tyCurrList	:= a_tyListTemp;
							eStatus			:= Done;

						ELSIF fbFileWriteList.udiStatus < 65534 THEN
							a_tyListTemp	:= a_tyCurrList;
							eStatus			:= Error;

							IF fbFileWriteList.udiStatus = 1900 THEN
								udiStatus	:= 10020;	//File Open Error While Adding & Editing
							ELSIF fbFileWriteList.udiStatus = 1901 THEN
								udiStatus	:= 10021;	//File Create Error While Adding & Editing
							ELSIF fbFileWriteList.udiStatus = 1903 THEN
								udiStatus	:= 10022;	//File Write Error While Adding & Editing
							ELSIF fbFileWriteList.udiStatus = 1904 THEN
								udiStatus	:= 10023;	//File Close Error While Adding & Editing
							ELSIF fbFileWriteList.udiStatus = 1914 THEN
								udiStatus	:= 10024;	//Directory Does Not Exist While Adding & Editing
							ELSE
								udiStatus	:= fbFileWriteList.udiStatus;
							END_IF
						END_IF

				END_CASE

			END_IF

		ProdRcpActReadCurrRcp:
			IF eStatus = Idle OR eStatus = Busy THEN

				eStatus	:= Busy;

				sStatTxt	:= a_sStatText[eStat];

				fbFileReadSingle(bEn := TRUE);
				IF fbFileReadSingle.udiStatus = 0 THEN
					eStatus			:= Done;

				ELSIF fbFileReadSingle.udiStatus < 65534 THEN
					eStatus		:= Error;

					IF fbFileReadSingle.udiStatus = 1900 THEN
						udiStatus	:= 10030;	//File Open Error While Reading Current Recipe
					ELSIF fbFileReadSingle.udiStatus = 1902 THEN
						udiStatus	:= 10031;	//File Read Error While Reading Current Recipe
					ELSIF fbFileReadSingle.udiStatus = 1904 THEN
						udiStatus	:= 10032;	//File Close Error While Reading Current Recipe
					ELSIF fbFileReadSingle.udiStatus = 1915 THEN
						eStatus			:= Done;
						bFileNotFound	:= TRUE;
					ELSE
						udiStatus	:= fbFileReadSingle.udiStatus;
					END_IF
				END_IF

			END_IF

		ProdRcpActWriteCurrRcpParam:
			IF eStatus = Idle OR eStatus = Busy THEN

				sStatTxt	:= a_sStatText[eStat];

				fbFileWriteSingle(bEn := TRUE);

				IF fbFileWriteSingle.udiStatus = 0 THEN
					a_tyCurrRcp[0]	:= p_tyCurrRcpWr;
					eStatus			:= Done;
				ELSIF fbFileWriteSingle.udiStatus < 65534 THEN
					eStatus			:= Error;

					IF fbFileWriteSingle.udiStatus = 1900 THEN
						udiStatus	:= 10033;	//File Open Error While Writing Current Recipe Parameter
					ELSIF fbFileWriteSingle.udiStatus = 1901 THEN
						udiStatus	:= 10034;	//File Create Error While Writing Current Recipe Parameter
					ELSIF fbFileWriteSingle.udiStatus = 1903 THEN
						udiStatus	:= 10035;	//File Write Error While Writing Current Recipe Parameter
					ELSIF fbFileWriteSingle.udiStatus = 1904 THEN
						udiStatus	:= 10036;	//File Close Error While Writing Current Recipe Parameter
					ELSIF fbFileWriteSingle.udiStatus = 1914 THEN
						udiStatus	:= 10037;	//Directory Does Not Exist Writing Current Recipe Parameter
					ELSE
						udiStatus	:= fbFileWriteSingle.udiStatus;
					END_IF
				END_IF

			END_IF

		ProdRcpActSaveList:
			IF eStatus = Idle OR eStatus = Busy THEN

				eStatus	:= Busy;

				sStatTxt	:= a_sStatText[eStat];

				CASE usiStep OF

					0:
						a_tyListTemp	:= a_tyCurrList;

						fbFileWriteList(bEn := TRUE);

						IF fbFileWriteList.udiStatus = 0 THEN
							eStatus			:= Done;

						ELSIF fbFileWriteList.udiStatus < 65534 THEN
							eStatus			:= Error;

							IF fbFileWriteList.udiStatus = 1900 THEN
								udiStatus	:= 10038;	//File Open Error While Saving List
							ELSIF fbFileWriteList.udiStatus = 1901 THEN
								udiStatus	:= 10039;	//File Create Error While Saving List
							ELSIF fbFileWriteList.udiStatus = 1903 THEN
								udiStatus	:= 10040;	//File Write Error While Saving List
							ELSIF fbFileWriteList.udiStatus = 1904 THEN
								udiStatus	:= 10041;	//File Close Error While Saving List
							ELSIF fbFileWriteList.udiStatus = 1914 THEN
								udiStatus	:= 10042;	//Directory Does Not Exist While Saving List
							ELSE
								udiStatus	:= fbFileWriteList.udiStatus;
							END_IF
						END_IF

				END_CASE

			END_IF

		ProdRcpActSort:
			IF eStatus = Idle OR eStatus = Busy THEN

				sStatTxt	:= a_sStatText[eStat];

				CASE usiStep OF

					0:

						FOR udi := 1 TO c_udiProdRcpMax DO
							IF p_sSearch <> '' THEN
								IF a_tyFilterList[udi].sRcpNm = '' THEN
									usiStep := 1;
									EXIT;
								ELSIF udi = c_udiProdRcpMax THEN
									iTotalRcp := UDINT_TO_INT(c_udiProdRcpMax);
									usiStep := 1;
									EXIT;
								ELSE
									iTotalRcp := iTotalRcp +1;
								END_IF
							ELSE
								IF a_tyCurrList[udi].sRcpNm = '' THEN
									usiStep := 1;
									EXIT;
								ELSIF udi = c_udiProdRcpMax THEN
									iTotalRcp := UDINT_TO_INT(c_udiProdRcpMax);
									usiStep := 1;
									EXIT;
								ELSE
									iTotalRcp := iTotalRcp +1;
								END_IF
							END_IF
						END_FOR

					1:
						IF p_sSearch <> '' THEN
							memcpy(ADR(a_tySortList),ADR(a_tyFilterList), SIZEOF(a_tyFilterList));
						ELSE
							memcpy(ADR(a_tySortList),ADR(a_tyCurrList), SIZEOF(a_tyCurrList));
						END_IF

						iSortCurrentOuterCntr	:= 0;
						iSortCurrentInnerCntr	:= 1 ;

						udiSortCurrenTotalCntr	:= 0;

						usiStep := 2;

					2:

						IF iSortCurrentOuterCntr < iTotalRcp THEN

							FOR iSortCurrentInnerCntr:= iSortCurrentOuterCntr+1 TO iTotalRcp-1 DO

								IF fRecipeNmCompare(ADR(a_tySortList[iSortCurrentOuterCntr+1].sRcpNm),ADR(a_tySortList[iSortCurrentInnerCntr+1].sRcpNm),SIZEOF(a_tySortList[1].sRcpNm),ADR(sDebug)) THEN

									memcpy(ADR(tyTempRecipe), ADR(a_tySortList[iSortCurrentOuterCntr+1]), SIZEOF(a_tySortList[1]));
									memcpy(ADR(a_tySortList[iSortCurrentOuterCntr+1]), ADR(a_tySortList[iSortCurrentInnerCntr+1]), SIZEOF(a_tySortList[1]));
									memcpy(ADR(a_tySortList[iSortCurrentInnerCntr+1]), ADR(tyTempRecipe), SIZEOF(a_tySortList[1]));

								END_IF

								udiSortCurrenTotalCntr	:= udiSortCurrenTotalCntr + 1;

							END_FOR

							iSortCurrentOuterCntr	:= iSortCurrentOuterCntr + 1;

						ELSE
							usiStep := 3;
						END_IF

					3:
						eStatus	:= Done;

				END_CASE

			END_IF

		ProdRcpActEndCharFilter:
			IF eStatus = Idle OR eStatus = Busy THEN

				sStatTxt	:= a_sStatText[eStat];

				fRecipeLastCharFilter(p_sScan , ADR(a_tyScanList) , ADR(a_tyCurrList) , SIZEOF(a_tyCurrList[1]) , ADR(a_tyCurrList[1].sRcpNm) , SIZEOF(a_tyCurrList[1].sRcpNm) , p_udiMax);

				eStatus	:= Done;

			END_IF

	END_CASE

END_ACTION
```

#### Act_Alarm.st - Do Not Change!!!
```iecst
(** 2019-03-25 **)
ACTION Act_Alarm:

	//Error
	IF EDGEPOS(eStatus = Error) THEN

		tyAlmData.sProgNm		:= p_sProgNm;
		tyAlmData.udiCode		:= udiStatus;
		tyAlmData.eSeverity		:= AlmSeverityError;
		tyAlmData.udiRunTime	:= tyAlmData.udiRunTime + 1;
		tyAlmData.bAlm			:= TRUE;
		tyAlmData.udiModuleNum  := udiModuleNum;
		g_sProdRcpProgNm		:= p_sProgNm;

		//Get Error Message
		IF tyAlmData.udiCode < 10000 OR tyAlmData.udiCode > 10099 THEN
			tyAlmData.sAlmMsg	:= 'Unknown';
			tyAlmData.sRcyMsg	:= 'Unknown';
		ELSE
			tyAlmData.sAlmMsg	:= a_tyAlmText[tyAlmData.udiCode].sAlmText;
			tyAlmData.sRcyMsg	:= a_tyAlmText[tyAlmData.udiCode].sRcyText;
		END_IF

		sStatTxt	:= tyAlmData.sAlmMsg;

	ELSIF bRstErr AND (tyAlmData.udiCode <> 0) THEN

		tyAlmData.udiCode	:= 0;
		tyAlmData.eSeverity	:= AlmSeverityNA;
		tyAlmData.sAlmMsg	:= '';
		tyAlmData.sRcyMsg	:= '';
		tyAlmData.bAlm		:= FALSE;

		sStatTxt	:= a_sStatText[eStat];

	END_IF

END_ACTION
```

#### InputRef.var - Do Not Change!!!
```iecst
(*2020-06-08*)
(**)
(*General*)
VAR
	p_eAct : REFERENCE TO eProdRcpAction;
	p_udiMax : REFERENCE TO UDINT;
	p_udiRstErr : REFERENCE TO UDINT;
END_VAR
(**)
(*Configuration*)
VAR
	p_dtCurrDT : REFERENCE TO DATE_AND_TIME;
	p_uiSortNo : REFERENCE TO UINT;
	p_sSearch : REFERENCE TO STRING[254];
	p_sScan : REFERENCE TO STRING[254];
	p_tyInfoIn : REFERENCE TO tyProdRcpParam;
	p_tyCurrRcpWr : REFERENCE TO tyProdRcpParam;
	p_sListFileName : REFERENCE TO STRING[80];
	p_sSingleFileName : REFERENCE TO STRING[80];
	p_sProgNm : REFERENCE TO STRING[15];
	p_bNtSettingsLoadDone : REFERENCE TO BOOL;
	p_bWidth2Prep : REFERENCE TO BOOL;
END_VAR
```

#### Local.var - Do Not Change!!!
```iecst
(*2023-02-13*)
(**)
(*Local Action, State & Status*)
VAR
	eAct : eProdRcpAction := ProdRcpActIdle;
	eStat : eProdRcpAction := ProdRcpActIdle;
	eStatus : eFBStatus := Idle;
	udiStatus : UDINT := 0;
	sStatTxt : STRING[200] := '';
	a_sStatText : ARRAY[0..50] OF STRING[200] := ['Idling','Creating Directory','Adding and Editing Files','Deleting Files','Get Info','Get List','Filtering Files','Loading Recipe','Adding Files','Editing Files','Reading Current Recipe','Writing Current Recipe Parameter','Saving Recipe List',38('')];
END_VAR
(**)
(*Local Alarm*)
VAR
	tyAlmData : tyAlmDat;
	a_tyAlmText : ARRAY[10000..10099] OF tyAlmTxt := [(sAlmText:='Create User Directory Error',sRcyText:='Unable To Create User Directory. Please Contact Nutek For A Possible Solution'),(sAlmText:='Create Product Recipe Directory Error',sRcyText:='Unable To Create Product Recipe Directory. Please Contact Nutek For A Possible Solution'),(sAlmText:='File Open Error While Adding & Editing',sRcyText:='An Error Was Encountered While Trying To Open File. Please Contact Nutek For A Possible Solution.'),(sAlmText:='File Create Error While Adding & Editing',sRcyText:='An Error Was Encountered While Trying To Create File. Please Contact Nutek For A Possible Solution.'),(sAlmText:='File Write Error While Adding & Editing',sRcyText:='An Error Was Encountered While Trying To Write File. Please Contact Nutek For A Possible Solution.'),(sAlmText:='File Close Error While Adding & Editing',sRcyText:='An Error Was Encountered While Trying To Close File. Please Contact Nutek For A Possible Solution.'),(sAlmText:='File Open Error While Deleting',sRcyText:='An Error Was Encountered While Trying To Open File. Please Contact Nutek For A Possible Solution.'),(sAlmText:='File Create Error While Deleting',sRcyText:='An Error Was Encountered While Trying To Create File. Please Contact Nutek For A Possible Solution.'),(sAlmText:='File Write Error While Deleting',sRcyText:='An Error Was Encountered While Trying To Write File. Please Contact Nutek For A Possible Solution.'),(sAlmText:='File Close Error While Deleting',sRcyText:='An Error Was Encountered While Trying To Close File. Please Contact Nutek For A Possible Solution.'),(sAlmText:='File Open Error While Getting List',sRcyText:='An Error Was Encountered While Trying To Open File. Please Contact Nutek For A Possible Solution.'),(sAlmText:='File Read Error While Getting List',sRcyText:='An Error Was Encountered While Trying To Read File. Please Contact Nutek For A Possible Solution.'),(sAlmText:='File Close Error While Getting List',sRcyText:='An Error Was Encountered While Trying To Close File. Please Contact Nutek For A Possible Solution.'),(sAlmText:='Directory Does Not Exist While Adding & Editing',sRcyText:='The Directory Does Not Exist.Please Contact Nutek For A Possible Solution.'),(sAlmText:='Directory Does Not Exist While Deleting',sRcyText:='The Directory Does Not Exist.Please Contact Nutek For A Possible Solution.'),(sAlmText:='File Open Error While Adding',sRcyText:='An Error Was Encountered While Trying To Open File. Please Contact Nutek For A Possible Solution.'),(sAlmText:='File Create Error While Adding',sRcyText:='An Error Was Encountered While Trying To Create File. Please Contact Nutek For A Possible Solution.'),(sAlmText:='File Write Error While Adding',sRcyText:='An Error Was Encountered While Trying To Write File. Please Contact Nutek For A Possible Solution.'),(sAlmText:='File Close Error While Adding',sRcyText:='An Error Was Encountered While Trying To Close File. Please Contact Nutek For A Possible Solution.'),(sAlmText:='Directory Does Not Exist While Adding',sRcyText:='The Directory Does Not Exist.Please Contact Nutek For A Possible Solution.'),(sAlmText:='File Open Error While Editing',sRcyText:='An Error Was Encountered While Trying To Open File. Please Contact Nutek For A Possible Solution.'),(sAlmText:='File Create Error While Editing',sRcyText:='An Error Was Encountered While Trying To Create File. Please Contact Nutek For A Possible Solution.'),(sAlmText:='File Write Error While Editing',sRcyText:='An Error Was Encountered While Trying To Write File. Please Contact Nutek For A Possible Solution.'),(sAlmText:='File Close Error While Editing',sRcyText:='An Error Was Encountered While Trying To Close File. Please Contact Nutek For A Possible Solution.'),(sAlmText:='Directory Does Not Exist While Editing',sRcyText:='The Directory Does Not Exist.Please Contact Nutek For A Possible Solution.'),(sAlmText:='File Open Error While Loading Current Recipe',sRcyText:='An Error Was Encountered While Trying To Open File. Please Contact Nutek For A Possible Solution.'),(sAlmText:='File Create Error While Loading Current Recipe',sRcyText:='An Error Was Encountered While Trying To Create File. Please Contact Nutek For A Possible Solution.'),(sAlmText:='File Write Error While Loading Current Recipe',sRcyText:='An Error Was Encountered While Trying To Write File. Please Contact Nutek For A Possible Solution.'),(sAlmText:='File Close Error While Loading Current Recipe',sRcyText:='An Error Was Encountered While Trying To Close File. Please Contact Nutek For A Possible Solution.'),(sAlmText:='Directory Does Not Exist While Loading Current Recipe',sRcyText:='The Directory Does Not Exist.Please Contact Nutek For A Possible Solution.'),(sAlmText:='File Open Error While Reading Current Recipe',sRcyText:='An Error Was Encountered While Trying To Open File. Please Contact Nutek For A Possible Solution.'),(sAlmText:='File Read Error While Reading Current Recipe',sRcyText:='An Error Was Encountered While Trying To Read File. Please Contact Nutek For A Possible Solution.'),(sAlmText:='File Close Error While Reading Current Recipe',sRcyText:='An Error Was Encountered While Trying To Close File. Please Contact Nutek For A Possible Solution.'),(sAlmText:='File Open Error While Writing Current Recipe Parameter',sRcyText:='An Error Was Encountered While Trying To Open File. Please Contact Nutek For A Possible Solution.'),(sAlmText:='File Create Error While Writing Current Recipe Parameter',sRcyText:='An Error Was Encountered While Trying To Create File. Please Contact Nutek For A Possible Solution.'),(sAlmText:='File Write Error While Writing Current Recipe Parameter',sRcyText:='An Error Was Encountered While Trying To Write File. Please Contact Nutek For A Possible Solution.'),(sAlmText:='File Close Error While Writing Current Recipe Parameter',sRcyText:='An Error Was Encountered While Trying To Close File. Please Contact Nutek For A Possible Solution.'),(sAlmText:='Directory Does Not Exist While Writing Current Recipe Parameter',sRcyText:='The Directory Does Not Exist.Please Contact Nutek For A Possible Solution.'),(sAlmText:='File Open Error While Writing Saving List',sRcyText:='An Error Was Encountered While Trying To Open File. Please Contact Nutek For A Possible Solution.'),(sAlmText:='File Create Error While Writing Saving List',sRcyText:='An Error Was Encountered While Trying To Create File. Please Contact Nutek For A Possible Solution.'),(sAlmText:='File Write Error While Writing Saving List',sRcyText:='An Error Was Encountered While Trying To Write File. Please Contact Nutek For A Possible Solution.'),(sAlmText:='File Close Error While Writing Saving List',sRcyText:='An Error Was Encountered While Trying To Close File. Please Contact Nutek For A Possible Solution.'),(sAlmText:='Directory Does Not Exist While Writing Saving List',sRcyText:='The Directory Does Not Exist.Please Contact Nutek For A Possible Solution.'),57(0)];
END_VAR
(**)
(*Local Output*)
VAR
	bNmExist : BOOL;
	bNmNotExist : BOOL;
	bNmEmpty : BOOL;
	bListFull : BOOL;
	a_tyCurrList : ARRAY[1..c_udiProdRcpMax] OF tyProdRcpParam;
	a_tyFilterList : ARRAY[1..c_udiProdRcpMax] OF tyProdRcpParam;
	a_tySortList : ARRAY[1..c_udiProdRcpMax] OF tyProdRcpParam;
	a_tyScanList : ARRAY[1..c_udiProdRcpMax] OF tyProdRcpParam;
	tyTempList : tyProdRcpParam;
	tyInfoOut : tyProdRcpParam;
	bFileNotFound : BOOL;
	a_tyCurrRcp : ARRAY[0..5] OF tyProdRcpParam;
END_VAR
(**)
(*Local Input*)
VAR
	udiRstErr : UDINT := 0;
	dtCurrDT : DATE_AND_TIME;
	sSearch : STRING[254] := '';
	sScan : STRING[254] := '';
	tyInfoIn : tyProdRcpParam;
	tyCurrRcpWr : tyProdRcpParam;
	sListFileName : STRING[80] := 'ProductRecipeList.dat';
	sSingleFileName : STRING[80] := 'ProductRecipe.dat';
	sProgNm : STRING[15] := 'ProdRcp';
	bNtSettingsLoadDone : BOOL := TRUE;
	bWidth2Prep : BOOL;
END_VAR
(**)
(*Local*)
VAR
	bRstErr : BOOL;
	udiRstErrOld : UDINT;
	bInitDone : BOOL;
	bInitialDone : BOOL;
	usiStep : USINT;
	udiAddStatus : UDINT;
	a_tyListTemp : ARRAY[1..c_udiProdRcpMax] OF tyProdRcpParam;
	fbDirCreate1 : fbDirCreate;
	fbDirCreate2 : fbDirCreate;
	fbFileReadList : fbFileFullRead;
	fbFileWriteList : fbFileFullWrite;
	fbFileReadSingle : fbFileFullRead;
	fbFileWriteSingle : fbFileFullWrite;
	fbFileLoadSingle : fbFileFullWrite;
	iFilterCtr : INT;
	udiModuleNum : UDINT := 4801;
END_VAR
```

### MpProdRcp.typ - Change By Project
```iecst
(*2019-04-28*)
(**)
(*Action*)

TYPE
	eMpProdRcpAction :
		(
		MpProdRcpActIdle,
		MpProdRcpActCreateDir,
		MpProdRcpActLoad,
		MpProdRcpActSave
		);
END_TYPE
```

### MpProdRcp.var - Change By Project
```iecst
(*2019-04-28*)
(**)
(*Action & State & Status*)
VAR
	p_MpProdRcpStat : UDINT;
	p_MpProdRcpStatus : UDINT;
	p_MpProdRcpStatTxt : UDINT;
END_VAR
(**)
(*Alarm*)
VAR
	p_MpProdRcpAlmData : UDINT;
END_VAR
(**)
(*Output*)
```

### Program Logical/MpProdRcp/MpProdRcp (IEC) - 1.00.0 - NtRecipe v5.00.0 , NtFileIO v5.00.0

#### InputRef.var
```iecst
(*2019-04-28*)
(**)
(*General*)
VAR
	p_eAct : REFERENCE TO eMpProdRcpAction;
	p_udiRstErr : REFERENCE TO UDINT;
END_VAR
(**)
(*Configuration*)
VAR
	pa_tyMpProdRcp : REFERENCE TO ARRAY[0..c_udiMpProdRcpMax] OF tyProdRcpParam;
	p_tyMpProdRcpMpLink : REFERENCE TO MpComIdentType;
	p_sPVName : REFERENCE TO STRING[100];
	p_sFileName : REFERENCE TO STRING[255];
	p_sProgNm : REFERENCE TO STRING[15];
	p_bNtSettingsLoadDone : REFERENCE TO BOOL;
END_VAR
```

#### InputRef_Link.var
```iecst
(*2019-04-28*)
(**)
VAR
	p_bLinkStartupRun : REFERENCE TO BOOL;
END_VAR
```

#### Local.var
```iecst
(*2019-04-30*)
(**)
(*Local Action, State & Status*)
VAR
	eAct : eMpProdRcpAction := MpProdRcpActIdle;
	eStat : eMpProdRcpAction := MpProdRcpActIdle;
	eStatus : eFBStatus := Idle;
	udiStatus : UDINT := 0;
	sStatTxt : STRING[200] := '';
	a_sStatText : ARRAY[0..50] OF STRING[200] := ['Idling','Creating Directory','Loading Mp Product Recipe','Saving Mp Product Recipe',47('')];
END_VAR
(**)
(*Local Alarm*)
VAR
	tyAlmData : tyAlmDat;
	a_tyAlmText : ARRAY[10000..10099] OF tyAlmTxt := [(sAlmText:='Create User Directory Error',sRcyText:='Unable To Create User Directory. Please Contact Nutek For A Possible Solution'),(sAlmText:='Create Product Recipe Directory Error',sRcyText:='Unable To Create Product Recipe Directory. Please Contact Nutek For A Possible Solution'),(sAlmText:='MpRecipeRegPar Error While Loading',sRcyText:='Unable To Register Parameter. Please Contact Nutek For A Possible Solution'),(sAlmText:='MpRecipeXml Error While Loading',sRcyText:='Unable To Handle Recipe In Xml. Please Contact Nutek For A Possible Solution'),(sAlmText:='MpRecipeRegPar Error While Saving',sRcyText:='Unable To Register Parameter. Please Contact Nutek For A Possible Solution'),(sAlmText:='MpRecipeXml Error While Saving',sRcyText:='Unable To Handle Recipe In Xml. Please Contact Nutek For A Possible Solution'),94((sAlmText:='',sRcyText:=''))];
END_VAR
(**)
(*Local Output*)
(**)
(*Local Input*)
VAR
	udiRstErr : UDINT := 0;
	a_tyMpProdRcp : ARRAY[0..c_udiMpProdRcpMax] OF tyProdRcpParam;
	tyMpProdRcpMpLink : MpComIdentType;
	sPVName : STRING[100] := 'MpProdRcp:a_tyMpProdRcp1';
	sFileName : STRING[255] := 'MpProductRecipe.xml';
	sProgNm : STRING[15] := 'MpProdRcp';
	bNtSettingsLoadDone : BOOL := TRUE;
END_VAR
(**)
(*Local*)
VAR
	bRstErr : BOOL;
	udiRstErrOld : UDINT;
	bInitDone : BOOL;
	bInitialDone : BOOL;
	usiStep : USINT;
	a_tyMpProdRcp1 : ARRAY[0..c_udiMpProdRcpMax] OF tyProdRcpParam;
	fbDirCreate1 : fbDirCreate;
	fbDirCreate2 : fbDirCreate;
	fbMpRecipeRegPar : MpRecipeRegPar;
	fbMpRecipeXml : MpRecipeXml;
END_VAR
VAR CONSTANT
	c_udiMpProdRcpMax : UDINT := 1999;
END_VAR
VAR
	udiModuleNum : UDINT := 5001;
END_VAR
```

#### Act_Action.st
```iecst
(** 2019-04-28 **)
ACTION Act_Action:

	//Reset Error
	IF (eStatus = Error) AND bRstErr THEN
		p_eAct	:= MpProdRcpActIdle;
		eStat	:= MpProdRcpActIdle;
	END_IF

	//Reset Done
	IF eStatus = Done AND p_eAct = MpProdRcpActIdle THEN
		eStat	:= MpProdRcpActIdle;
	END_IF

	//Set p_eAct
	IF eStatus = Idle THEN
		eStat	:= p_eAct;
	END_IF

END_ACTION
```

#### Act_Alarm.st
```iecst
(** 2019-04-28 **)
ACTION Act_Alarm:

	//Error
	IF EDGEPOS(eStatus = Error) THEN

		tyAlmData.sProgNm		:= p_sProgNm;
		tyAlmData.udiCode		:= udiStatus;
		tyAlmData.eSeverity		:= AlmSeverityError;
		tyAlmData.udiRunTime	:= tyAlmData.udiRunTime + 1;
		tyAlmData.bAlm			:= TRUE;
		tyAlmData.udiModuleNum  := udiModuleNum;
		g_sMpProdRcpProgNm		:= p_sProgNm;

		//Get Error Message
		IF tyAlmData.udiCode < 10000 OR tyAlmData.udiCode > 10099 THEN
			tyAlmData.sAlmMsg	:= 'Unknown';
			tyAlmData.sRcyMsg	:= 'Unknown';
		ELSE
			tyAlmData.sAlmMsg	:= a_tyAlmText[tyAlmData.udiCode].sAlmText;
			tyAlmData.sRcyMsg	:= a_tyAlmText[tyAlmData.udiCode].sRcyText;
		END_IF

		sStatTxt	:= tyAlmData.sAlmMsg;

	ELSIF bRstErr AND (tyAlmData.udiCode <> 0) THEN

		tyAlmData.udiCode	:= 0;
		tyAlmData.eSeverity	:= AlmSeverityNA;
		tyAlmData.sAlmMsg	:= '';
		tyAlmData.sRcyMsg	:= '';
		tyAlmData.bAlm			:= FALSE;
		sStatTxt	:= a_sStatText[eStat];

	END_IF

END_ACTION
```

#### Act_InitGlobal.st
```iecst
(** 2019-04-28 **)
ACTION Act_InitGlobal:

	(* Always Change If Project Change *)

	//Pass Data To Link
	p_bLinkStartupRun ACCESS p_StartupRun;

	//Pass Data To Internal Use
	p_udiRstErr ACCESS p_RstErrReset;
	pa_tyMpProdRcp ACCESS p_ProdRcpCurrList;
	p_sPVName ACCESS p_NtParamMpProdRcpPVNm;
	p_sFileName ACCESS p_NtParamMpProdRcpFileNm;
	p_sProgNm ACCESS p_NtParamMpProdRcpProgNm;
	p_bNtSettingsLoadDone ACCESS p_StartupNtSettingsLoadDone;

	(* Always Change If Project Change *)

END_ACTION
```

#### Act_Initial.st
```iecst
(** 2019-04-28 **)
ACTION Act_Initial:

	//Initial
	sStatTxt	:= a_sStatText[eStat];

	fbDirCreate1.sDevice	:= 'F';
	fbDirCreate1.sDirName	:= 'User';
	fbDirCreate1(bEn := FALSE);

	fbDirCreate2.sDevice	:= 'User';
	fbDirCreate2.sDirName	:= 'ProductRecipeXml';
	fbDirCreate2(bEn := FALSE);

	tyMpProdRcpMpLink	:= gRecipeXml;

	fbMpRecipeRegPar.MpLink	:= ADR(p_tyMpProdRcpMpLink);
	fbMpRecipeRegPar.PVName	:= ADR(p_sPVName);
	fbMpRecipeRegPar(Enable := FALSE);

	fbMpRecipeXml.MpLink		:= ADR(p_tyMpProdRcpMpLink);
	fbMpRecipeXml.DeviceName	:= ADR('MpProdRcp');
	fbMpRecipeXml.FileName		:= ADR(p_sFileName);
	fbMpRecipeXml(Enable := FALSE);

END_ACTION
```

#### Act_InitLocal.st
```iecst
(** 2019-04-28 **)
ACTION Act_InitLocal:

	//Input Reference Link To Local Variable
	p_eAct ACCESS ADR(eAct);
	p_udiRstErr ACCESS ADR(udiRstErr);
	pa_tyMpProdRcp ACCESS ADR(a_tyMpProdRcp);
	p_tyMpProdRcpMpLink ACCESS ADR(tyMpProdRcpMpLink);
	p_sPVName ACCESS ADR(sPVName);
	p_sFileName ACCESS ADR(sFileName);
	p_sProgNm ACCESS ADR(sProgNm);
	p_bNtSettingsLoadDone ACCESS ADR(bNtSettingsLoadDone);

END_ACTION
```

#### Act_Link.st
```iecst
(** 2019-04-28 **)
ACTION Act_Link:

END_ACTION
```

#### Act_LinkAction.st
```iecst
(** 2019-04-28 **)
ACTION Act_LinkAction:

	IF p_bLinkStartupRun = TRUE THEN
		p_eAct ACCESS p_StartupMpProdRcpAct;
	ELSE
		p_eAct ACCESS p_UIMpProdRcpAct;
	END_IF

END_ACTION
```

#### Act_Main.st
```iecst
(** 2019-04-28 **)
ACTION Act_Main:

	//Main
	CASE eStat OF

		MpProdRcpActIdle:
			IF eStatus <> Idle THEN	//Reset Data
				//Private
				fbDirCreate1(bEn := FALSE);
				fbDirCreate2(bEn := FALSE);
				fbMpRecipeRegPar(Enable := FALSE);
				fbMpRecipeXml(Enable := FALSE);
				usiStep			:= 0;

				sStatTxt	:= a_sStatText[eStat];

			END_IF

			eStatus	:= Idle;

		MpProdRcpActCreateDir:
			IF eStatus = Idle OR eStatus = Busy THEN

				eStatus	:= Busy;

				sStatTxt	:= a_sStatText[eStat];

				CASE usiStep OF
					0:
						fbDirCreate1(bEn := TRUE);
						IF fbDirCreate1.udiStatus = 0 THEN
							usiStep	:= 1;
						ELSIF fbDirCreate1.udiStatus < 65534 THEN
							eStatus		:= Error;

							IF fbDirCreate1.udiStatus = 1908 THEN
								udiStatus	:= 10000;	//Create User Directory Error
							ELSE
								udiStatus	:= fbDirCreate1.udiStatus;
							END_IF
						END_IF

					1:
						fbDirCreate2(bEn := TRUE);
						IF fbDirCreate2.udiStatus = 0 THEN
							eStatus	:= Done;
						ELSIF fbDirCreate2.udiStatus < 65534 THEN
							eStatus		:= Error;

							IF fbDirCreate2.udiStatus = 1908 THEN
								udiStatus	:= 10001;	//Create Product Recipe Directory Error
							ELSE
								udiStatus	:= fbDirCreate2.udiStatus;
							END_IF
						END_IF

				END_CASE

			END_IF

		MpProdRcpActLoad:
			IF eStatus = Idle OR eStatus = Busy THEN

				eStatus	:= Busy;

				sStatTxt	:= a_sStatText[eStat];

				CASE usiStep OF
					0:
						fbMpRecipeRegPar(Enable := TRUE);

						IF (fbMpRecipeRegPar.Active = TRUE) AND (fbMpRecipeRegPar.StatusID = 0) THEN
							usiStep	:= 1;
						ELSIF fbMpRecipeRegPar.StatusID <> 0 THEN
							eStatus		:= Error;
							udiStatus	:= 10002;	//MpRecipeRegPar Error While Loading
						END_IF

					1:
						fbMpRecipeXml.Load	:= TRUE;
						fbMpRecipeXml.Save	:= FALSE;
						fbMpRecipeXml(Enable := TRUE);

						IF (fbMpRecipeXml.Active = TRUE) AND (fbMpRecipeXml.CommandDone = TRUE) AND (fbMpRecipeXml.StatusID = 0) THEN
							eStatus	:= Done;
							pa_tyMpProdRcp	:= a_tyMpProdRcp1;
						ELSIF fbMpRecipeXml.StatusID <> 0 THEN
							eStatus		:= Error;
							udiStatus	:= 10003;	//MpRecipeXml Error While Loading
						END_IF

				END_CASE

			END_IF

		MpProdRcpActSave:
			IF eStatus = Idle OR eStatus = Busy THEN

				eStatus	:= Busy;

				sStatTxt	:= a_sStatText[eStat];

				CASE usiStep OF
					0:
						a_tyMpProdRcp1	:= pa_tyMpProdRcp;
						fbMpRecipeRegPar(Enable := TRUE);

						IF (fbMpRecipeRegPar.Active = TRUE) AND (fbMpRecipeRegPar.StatusID = 0) THEN
							usiStep	:= 1;
						ELSIF fbMpRecipeRegPar.StatusID <> 0 THEN
							eStatus		:= Error;
							udiStatus	:= 10004;	//MpRecipeRegPar Error While Saving
						END_IF

					1:
						fbMpRecipeXml.Load	:= FALSE;
						fbMpRecipeXml.Save	:= TRUE;
						fbMpRecipeXml(Enable := TRUE);

						IF (fbMpRecipeXml.Active = TRUE) AND (fbMpRecipeXml.CommandDone = TRUE) AND (fbMpRecipeXml.StatusID = 0) THEN
							eStatus	:= Done;
						ELSIF fbMpRecipeXml.StatusID <> 0 THEN
							eStatus		:= Error;
							udiStatus	:= 10005;	//MpRecipeXml Error While Saving
						END_IF

				END_CASE

			END_IF

	END_CASE

END_ACTION
```

#### Act_RstErr.st
```iecst
(** 2019-04-28 **)
ACTION Act_RstErr:

	IF p_udiRstErr <> udiRstErrOld THEN
		bRstErr			:= TRUE;
		udiRstErrOld	:= p_udiRstErr;
	ELSE
		bRstErr			:= FALSE;
	END_IF

END_ACTION
```

#### Cyclic.st
```iecst
(** 2019-04-28 **)
PROGRAM _CYCLIC

	IF bInitDone = FALSE THEN
		bInitDone	:= TRUE;

		Act_InitLocal;
		Act_InitGlobal;

	ELSIF bInitialDone = FALSE THEN
		IF p_bNtSettingsLoadDone = TRUE THEN
			bInitialDone	:= TRUE;

			Act_Initial;
		END_IF

	ELSE

		Act_RstErr;
		Act_LinkAction;
		Act_Action;
		Act_Link;
		Act_Main;
		Act_Alarm;

	END_IF

END_PROGRAM
```

#### Init.st
```iecst
(** 2019-04-28 **)
PROGRAM _INIT

	(* Always Change If Project Change *)

	//Pass Address To Global Address For External Use
	//Action, State & Status
	p_MpProdRcpStat		:= ADR(eStat);
	p_MpProdRcpStatus	:= ADR(eStatus);
	p_MpProdRcpStatTxt	:= ADR(sStatTxt);

	//Alarm
	p_MpProdRcpAlmData	:= ADR(tyAlmData);

	//Output

	(* Always Change If Project Change *)

END_PROGRAM
```

### McParam.var - Change By Project
```iecst
(*2019-04-17*)
(**)
(*Action & State & Status*)
VAR
	p_McParamStat : UDINT;
	p_McParamStatus : UDINT;
	p_McParamStatTxt : UDINT;
END_VAR
(**)
(*Alarm*)
VAR
	p_McParamAlmData : UDINT;
END_VAR
(**)
(*Output*)
VAR
	p_McParamFileNotFound : UDINT;
END_VAR
(**)
VAR
	p_McParamCurr : UDINT;
END_VAR
(**)
VAR
	p_McParamLFOnline : UDINT;
	p_McParamLFIPAddr : UDINT;
END_VAR
(**)
VAR
	p_McParamMcNm : UDINT;
	p_McParamWidthAtHmPos : UDINT;
	p_McParamWidthOffset : UDINT;
	p_McParamSSaverEn : UDINT;
	p_McParamSSaverTm : UDINT;
	p_McParamConvInitTm : UDINT;
	p_McParamTranInErrDlyTm : UDINT;
	p_McParamTranOutErrDlyTm : UDINT;
	p_McParamDefaultMcMod : UDINT;
	p_McParamDefaultFlippedBrd : UDINT;
	p_McParamAutoStepEn : UDINT;
	p_McParamAWDis : UDINT;
	p_McParamVSMEMAEn : UDINT;
	p_McParamMnlAccDat : UDINT;
	p_McParamChgParamEn : UDINT;
	p_McParamHermesRmtEn : UDINT;
END_VAR
(**)
VAR
	p_McParamLang : UDINT;
END_VAR
(**)
VAR
	p_McParamLFEn : UDINT;
	p_McParamLCSLFEn : UDINT;
	p_McParamLCSReqRcpEn : UDINT;
	p_McParamLCSManageRcpEn : UDINT;
	p_McParamLCSLiveDatEn : UDINT;
	p_McParamSectionLeader : UDINT;
	p_McParamUSWidthChkEn : UDINT;
	p_McParamDSWidthChkEn : UDINT;
END_VAR
(**)
VAR
	p_McParamConvLftSenAntiGap : UDINT;
	p_McParamConvLftSenOnTm : UDINT;
	p_McParamConvLftSenOffTm : UDINT;
	p_McParamConvRgtSenAntiGap : UDINT;
	p_McParamConvRgtSenOnTm : UDINT;
	p_McParamConvRgtSenOffTm : UDINT;
END_VAR
(**)
VAR
	p_McParamUSCommMod : UDINT;
	p_McParamUSSMEMAParam : UDINT;
	p_McParamUSSMEMASelection : UDINT;
	p_McParamUBAStatSetGd : UDINT;
END_VAR
(**)
VAR
	p_McParamDSCommMod : UDINT;
	p_McParamDSSMEMAParam : UDINT;
	p_McParamDSSMEMASelection : UDINT;
	p_McParamDBAStatSetGd : UDINT;
END_VAR
(**)
VAR
	p_McParamUSComm2Mod : UDINT;
	p_McParamUSSMEMA2Param : UDINT;
	p_McParamUSSMEMA2Selection : UDINT;
	p_McParamUBAStat2SetGd : UDINT;
END_VAR
(*  *)
VAR
	p_McParamDSComm2Mod : UDINT;
	p_McParamDSSMEMA2Param : UDINT;
	p_McParamDSSMEMA2Selection : UDINT;
	p_McParamDBAStat2SetGd : UDINT;
END_VAR
(**)
VAR
	p_McParamStopperDis : UDINT;
	p_McParamClampDis : UDINT;
	p_McParamInShutterDis : UDINT;
	p_McParamOutShutterDis : UDINT;
END_VAR
(**)
VAR
	p_McParamStopperAtLftPos : UDINT;
	p_McParamStopperAtRgtPos : UDINT;
END_VAR
(**)
VAR
	p_McParamLFLeaderMc : UDINT;
	p_McParamLFMcIdxBeforeOven : UDINT;
	p_McParamLFMcIdxAfterOven : UDINT;
	p_McParamLFMcIdxBeforeOven2 : UDINT;
	p_McParamLFMcIdxAfterOven2 : UDINT;
END_VAR
(**)
VAR
	p_McParamNetworkMod : UDINT;
	p_McParamLFSeqStayActive : UDINT;
	p_McParamLFBuzMute : UDINT;
	p_McParamDBAOnWOAlign : UDINT;
END_VAR
(**)
```

### McParam.typ - Change By Project
```iecst
(*2019-05-04*)
(**)
(*Action*)

TYPE
	eMcParamAction :
		(
		McParamActIdle,
		McParamActCreateDir,
		McParamActRead,
		McParamActWrite
		);
END_TYPE

(**)
(*Data*)

TYPE
	tyMcParam : 	STRUCT
		a_bLFOnline : ARRAY[1..c_diLFClntNum]OF BOOL;
		a_sLFIPAddr : ARRAY[1..c_diLFClntNum]OF STRING[15];
		sMcNm : STRING[30] := 'Inverter';
		diWidthAtHmPosInUM : DINT := 256800;
		sIPAddr : STRING[15] := '192.168.0.40';
		sSubnetMask : STRING[15] := '255.255.255.0';
		eNetworkMod : eNetworkConfigMod := SetIPManually;
		bSSaverEn : BOOL := FALSE;
		uiSSaverTmInSec : UINT := 1800;
		diConvInitTmInMS : DINT := 6000;
		diTranInErrDlyTmInMS : DINT := 12000;
		diTranOutErrDlyTmInMS : DINT := 12000;
		diStopperAtLftPos : DINT := 99500;
		diStopperAtRgtPos : DINT := 0;
		usiDefaultMcMod : USINT := 0;
		usiDefaultFlippedBrd : USINT := 0;
		bAutoStepEn : BOOL := FALSE;
		bAWDis : BOOL := FALSE;
		bVSMEMAEn : BOOL := FALSE;
		bMnlAccDat : BOOL := FALSE;
		bChgParamEn : BOOL := FALSE;
		bHermesRmtEn : BOOL := FALSE;
		bHermesSvyEn : BOOL := FALSE;
		bClampDis : BOOL := FALSE;
		bStopperDis : BOOL := FALSE;
		bInShutterDis : BOOL := FALSE;
		bOutShutterDis : BOOL := FALSE;
		usiLang : USINT := 0;
		bLFEn : BOOL := FALSE;
		bLCSLFEn : BOOL := FALSE;
		bLCSReqRcpEn : BOOL := FALSE;
		bLCSManageRcpEn : BOOL := FALSE;
		bLCSLiveDatEn : BOOL := FALSE;
		bSectionLeader : BOOL := FALSE;
		bUSWidthChkEn : BOOL := FALSE;
		bDSWidthChkEn : BOOL := FALSE;
		tyConvLftSenAntiGapDly : tyAntiGapDly;
		tyConvRgtSenAntiGapDly : tyAntiGapDly;
		eUSComm : eMcSetCommMod := McSetCommModSMEMA;
		tyUSCommSMEMA : tySMEMAParam := (eSelection:=SMEMASelIPC9851,bStatSigSetGd:=FALSE);
		eDSComm : eMcSetCommMod := McSetCommModSMEMA;
		tyDSCommSMEMA : tySMEMAParam := (eSelection:=SMEMASelIPC9851,bStatSigSetGd:=FALSE);
		eUSComm2 : eMcSetCommMod := McSetCommModSMEMA;
		tyUSCommSMEMA2 : tySMEMAParam := (eSelection:=SMEMASelIPC9851,bStatSigSetGd:=FALSE);
		eDSComm2 : eMcSetCommMod := McSetCommModSMEMA;
		tyDSCommSMEMA2 : tySMEMAParam := (eSelection:=SMEMASelIPC9851,bStatSigSetGd:=FALSE);
		bLFLeaderMc : BOOL := FALSE;
		diLFMcIdxBeforeOven : DINT := 1;
		diLFMcIdxAfterOven : DINT := 1;
		diLFMcIdxBeforeOven2 : DINT := 1;
		diLFMcIdxAfterOven2 : DINT := 1;
		diWidthOffsetInUM : DINT := 0;
		bAutoLogoutEn : BOOL := FALSE;
		diAutoLogoutTmInSec : DINT := 1800000;
		bLFSeqStayActive : BOOL := FALSE;
		bLFBuzMute : BOOL := FALSE;
		bDBAOnWOAlign : BOOL := FALSE;
	END_STRUCT;
END_TYPE

(**)

TYPE
	tyAntiGapDly : 	STRUCT
		diSigOnTm : DINT;
		diSigOffTm : DINT;
	END_STRUCT;
	eMcSetCommMod :
		(
		McSetCommModSMEMA,
		McSetCommModHermes
		);
END_TYPE
```

### Program Logical/McParam/McParam (IEC)

#### InputRef.var
```iecst
(*2019-03-25*)
(**)
(*General*)
VAR
	p_eAct : REFERENCE TO eMcParamAction;
	p_udiRstErr : REFERENCE TO UDINT;
END_VAR
(**)
(*Configuration*)
VAR
	p_sFileName : REFERENCE TO STRING[80];
	p_tyMcParamWr : REFERENCE TO tyMcParam;
	p_sProgNm : REFERENCE TO STRING[15];
	p_bNtSettingsLoadDone : REFERENCE TO BOOL;
END_VAR
```

#### Local.var
```iecst
(*2019-04-30*)
(**)
(*Local Action, State & Status*)
VAR
	eAct : eMcParamAction := McParamActIdle;
	eStat : eMcParamAction := McParamActIdle;
	eStatus : eFBStatus := Idle;
	udiStatus : UDINT := 0;
	sStatTxt : STRING[200] := '';
	a_sStatText : ARRAY[0..50] OF STRING[200] := ['Idling','Creating Directory','Reading Files','Writing Files',47('')];
END_VAR
(**)
(*Local Alarm*)
VAR
	tyAlmData : tyAlmDat;
	a_tyAlmText : ARRAY[10000..10099] OF tyAlmTxt := [(sAlmText:='Create User Directory Error',sRcyText:='Unable To Create User Directory. Please Contact Nutek For A Possible Solution'),(sAlmText:='Create Machine Parameter Directory Error',sRcyText:='Unable To Create Machine Parameter Directory. Please Contact Nutek For A Possible Solution'),(sAlmText:='File Open Error While Writing',sRcyText:='An Error Was Encountered While Trying To Open File. Please Contact Nutek For A Possible Solution.'),(sAlmText:='File Create Error While Writing',sRcyText:='An Error Was Encountered While Trying To Create File. Please Contact Nutek For A Possible Solution.'),(sAlmText:='File Write Error',sRcyText:='An Error Was Encountered While Trying To Write File. Please Contact Nutek For A Possible Solution.'),(sAlmText:='File Close Error While Writing',sRcyText:='An Error Was Encountered While Trying To Close File. Please Contact Nutek For A Possible Solution.'),(sAlmText:='File Open Error While Reading',sRcyText:='An Error Was Encountered While Trying To Open File. Please Contact Nutek For A Possible Solution.'),(sAlmText:='File Read Error',sRcyText:='An Error Was Encountered While Trying To Read File. Please Contact Nutek For A Possible Solution.'),(sAlmText:='File Close Error While Reading',sRcyText:='An Error Was Encountered While Trying To Close File. Please Contact Nutek For A Possible Solution.'),(sAlmText:='Directory Does Not Exist While Writing',sRcyText:='The Directory Does Not Exist.Please Contact Nutek For A Possibe Solution.'),90(0)];
END_VAR
(**)
(*Local Output*)
VAR
	tyMcParamCurr : tyMcParam;
	bFileNotFound : BOOL;
END_VAR
(**)
(*Local Input*)
VAR
	udiRstErr : UDINT := 0;
	sFileName : STRING[80] := 'MachineParameter.dat';
	tyMcParamWr : tyMcParam;
	sProgNm : STRING[15] := 'McParam';
	bNtSettingsLoadDone : BOOL := TRUE;
END_VAR
(**)
(*Local*)
VAR
	bRstErr : BOOL;
	udiRstErrOld : UDINT;
	bInitDone : BOOL;
	bInitialDone : BOOL;
	usiStep : USINT;
	tyMcParamTemp : tyMcParam;
	fbDirCreate1 : fbDirCreate;
	fbDirCreate2 : fbDirCreate;
	fbFileRead1 : fbFileFullRead;
	fbFileWrite1 : fbFileFullWrite;
	fbFileWrite2 : fbFileFullWrite;
	udiModuleNum : UINT := 5251;
END_VAR
```

#### Act_Action.st
```iecst
(** 2019-03-25 **)
ACTION Act_Action:

	//Reset Error
	IF (eStatus = Error) AND bRstErr THEN
		p_eAct	:= McParamActIdle;
		eStat	:= McParamActIdle;
	END_IF

	//Reset Done
	IF eStatus = Done AND p_eAct = McParamActIdle THEN
		eStat	:= McParamActIdle;
	END_IF

	//Set p_eAct
	IF eStatus = Idle THEN
		eStat	:= p_eAct;
	END_IF

END_ACTION
```

#### Act_Alarm.st
```iecst
(** 2019-03-25 **)
ACTION Act_Alarm:

	//Error
	IF EDGEPOS(eStatus = Error) THEN

		tyAlmData.sProgNm		:= p_sProgNm;
		tyAlmData.udiCode		:= udiStatus;
		tyAlmData.eSeverity		:= AlmSeverityError;
		tyAlmData.udiRunTime	:= tyAlmData.udiRunTime + 1;
		tyAlmData.bAlm			:= TRUE;
		tyAlmData.udiModuleNum  := udiModuleNum;
		g_sMcParamProgNm		:= p_sProgNm;

		//Get Error Message
		IF tyAlmData.udiCode < 10000 OR tyAlmData.udiCode > 10099 THEN
			tyAlmData.sAlmMsg	:= 'Unknown';
			tyAlmData.sRcyMsg	:= 'Unknown';
		ELSE
			tyAlmData.sAlmMsg	:= a_tyAlmText[tyAlmData.udiCode].sAlmText;
			tyAlmData.sRcyMsg	:= a_tyAlmText[tyAlmData.udiCode].sRcyText;
		END_IF

		sStatTxt	:= tyAlmData.sAlmMsg;

	ELSIF bRstErr AND (tyAlmData.udiCode <> 0) THEN

		tyAlmData.udiCode	:= 0;
		tyAlmData.eSeverity	:= AlmSeverityNA;
		tyAlmData.sAlmMsg	:= '';
		tyAlmData.sRcyMsg	:= '';
		tyAlmData.bAlm			:= FALSE;
		sStatTxt	:= a_sStatText[eStat];

	END_IF

END_ACTION
```

#### Act_InitGlobal.st
```iecst
(** 2019-03-25 **)
ACTION Act_InitGlobal:

	(* Always Change If Project Change *)

	//Pass Data To Link
	p_bLinkStartupRun ACCESS p_StartupRun;

	//Pass Data To Internal Use
	p_udiRstErr ACCESS p_RstErrReset;
	p_sFileName ACCESS p_NtParamMcParamFileNm;
	p_tyMcParamWr ACCESS p_UIMcParamWr;
	p_sProgNm ACCESS p_NtParamMcParamProgNm;
	p_bNtSettingsLoadDone ACCESS p_StartupNtSettingsLoadDone;

	(* Always Change If Project Change *)

END_ACTION
```

#### Act_Initial.st
```iecst
(** 2019-01-15 **)
ACTION Act_Initial:

	//Initial
	sStatTxt	:= a_sStatText[eStat];

	fbDirCreate1.sDevice	:= 'F';
	fbDirCreate1.sDirName	:= 'User';
	fbDirCreate1(bEn := FALSE);

	fbDirCreate2.sDevice	:= 'User';
	fbDirCreate2.sDirName	:= 'MachineParameter';
	fbDirCreate2(bEn := FALSE);

	fbFileRead1.sDevice			:= 'McParam';
	fbFileRead1.sFile			:= p_sFileName;
	fbFileRead1.udiOffset		:= 0;
	fbFileRead1.p_Dest			:= ADR(tyMcParamCurr);
	fbFileRead1.udiLen			:= SIZEOF(tyMcParamCurr);
	fbFileRead1(bEn := FALSE);

	fbFileWrite1.sDevice		:= 'McParam';
	fbFileWrite1.sFile			:= p_sFileName;
	fbFileWrite1.udiOffset		:= 0;
	fbFileWrite1.p_Src			:= ADR(p_tyMcParamWr);
	fbFileWrite1.udiLen			:= SIZEOF(p_tyMcParamWr);
	fbFileWrite1.udiOption		:= 0;
	fbFileWrite1(bEn := FALSE);

	fbFileWrite2.sDevice		:= 'McParam';
	fbFileWrite2.sFile			:= p_sFileName;
	fbFileWrite2.udiOffset		:= 0;
	fbFileWrite2.p_Src			:= ADR(tyMcParamTemp);
	fbFileWrite2.udiLen			:= SIZEOF(tyMcParamTemp);
	fbFileWrite2.udiOption		:= 0;
	fbFileWrite2(bEn := FALSE);

END_ACTION
```

#### Act_InitLocal.st
```iecst
(** 2019-03-25 **)
ACTION Act_InitLocal:

	//Input Reference Link To Local Variable
	p_eAct ACCESS ADR(eAct);
	p_udiRstErr ACCESS ADR(udiRstErr);
	p_sFileName ACCESS ADR(sFileName);
	p_tyMcParamWr ACCESS ADR(tyMcParamWr);
	p_sProgNm ACCESS ADR(sProgNm);
	p_bNtSettingsLoadDone ACCESS ADR(bNtSettingsLoadDone);

END_ACTION
```

#### Act_Link.st
```iecst
(** 2019-03-29 **)
ACTION Act_Link:

	    //new for Hermes 1.3
	IF p_bRmtHermesWriteConfig OR p_bSvyHermesWriteConfig THEN
		p_tyMcParamWr.sMcNm := p_tyHermesConfigurationWr.tySvyParam.sMachineId;
	END_IF

END_ACTION
```

#### Act_LinkAction.st
```iecst
(** 2019-03-29 **)
ACTION Act_LinkAction:

	IF p_bLinkStartupRun = TRUE THEN
		p_eAct ACCESS p_StartupMcParamAct;
	ELSE
		p_eAct ACCESS p_UIMcParamAct;
	END_IF

END_ACTION
```

#### Act_Main.st
```iecst
(** 2019-01-10 **)
ACTION Act_Main:

	//Main
	CASE eStat OF

		McParamActIdle:
			IF eStatus <> Idle THEN	//Reset Data
				//Private
				fbDirCreate1(bEn := FALSE);
				fbDirCreate2(bEn := FALSE);
				fbFileRead1(bEn := FALSE);
				fbFileWrite1(bEn := FALSE);
				fbFileWrite2(bEn := FALSE);
				usiStep	:= 0;

				bFileNotFound	:= FALSE;

				sStatTxt	:= a_sStatText[eStat];

			END_IF

			eStatus	:= Idle;

		McParamActCreateDir:
			IF eStatus = Idle OR eStatus = Busy THEN

				eStatus	:= Busy;

				sStatTxt	:= a_sStatText[eStat];

				CASE usiStep OF
					0:
						fbDirCreate1(bEn := TRUE);
						IF fbDirCreate1.udiStatus = 0 THEN
							usiStep	:= 1;
						ELSIF fbDirCreate1.udiStatus < 65534 THEN
							eStatus		:= Error;

							IF fbDirCreate1.udiStatus = 1908 THEN
								udiStatus	:= 10000;	//Create User Directory Error
							ELSE
								udiStatus	:= fbDirCreate1.udiStatus;
							END_IF
						END_IF

					1:
						fbDirCreate2(bEn := TRUE);
						IF fbDirCreate2.udiStatus = 0 THEN
							eStatus	:= Done;
						ELSIF fbDirCreate2.udiStatus < 65534 THEN
							eStatus		:= Error;

							IF fbDirCreate2.udiStatus = 1908 THEN
								udiStatus	:= 10001;	//Create Machine Parameter Directory Error
							ELSE
								udiStatus	:= fbDirCreate2.udiStatus;
							END_IF
						END_IF

				END_CASE

			END_IF

		McParamActWrite:
			IF eStatus = Idle OR eStatus = Busy THEN

				eStatus	:= Busy;

				sStatTxt	:= a_sStatText[eStat];

				fbFileWrite1(bEn := TRUE);

				IF fbFileWrite1.udiStatus = 0 THEN
					tyMcParamCurr	:= p_tyMcParamWr;
					eStatus			:= Done;
				ELSIF fbFileWrite1.udiStatus < 65534 THEN
					eStatus			:= Error;

					IF fbFileWrite1.udiStatus = 1900 THEN
						udiStatus	:= 10002;	//File Open Error While Writing
					ELSIF fbFileWrite1.udiStatus = 1901 THEN
						udiStatus	:= 10003;	//File Create Error While Writing
					ELSIF fbFileWrite1.udiStatus = 1903 THEN
						udiStatus	:= 10004;	//File Write Error
					ELSIF fbFileWrite1.udiStatus = 1904 THEN
						udiStatus	:= 10005;	//File Close Error While Writing
					ELSIF fbFileWrite1.udiStatus = 1914 THEN
						udiStatus	:= 10009;	//Directory Does Not Exist While Writing
					ELSE
						udiStatus	:= fbFileWrite1.udiStatus;
					END_IF
				END_IF

			END_IF

		McParamActRead:
			IF eStatus = Idle OR eStatus = Busy THEN

				eStatus	:= Busy;

				sStatTxt	:= a_sStatText[eStat];

				fbFileRead1(bEn := TRUE);
				IF fbFileRead1.udiStatus = 0 THEN
					eStatus			:= Done;
				ELSIF fbFileRead1.udiStatus < 65534 THEN
					eStatus		:= Error;

					IF fbFileRead1.udiStatus = 1900 THEN
						udiStatus	:= 10006;	//File Open Error While Reading
					ELSIF fbFileRead1.udiStatus = 1902 THEN
						udiStatus	:= 10007;	//File Read Error
					ELSIF fbFileRead1.udiStatus = 1904 THEN
						udiStatus	:= 10008;	//File Close Error While Reading
					ELSIF fbFileRead1.udiStatus = 1915 THEN
						eStatus			:= Done;
						bFileNotFound	:= TRUE;
					ELSE
						udiStatus	:= fbFileRead1.udiStatus;
					END_IF
				END_IF

			END_IF

	END_CASE

END_ACTION
```

#### Act_RstErr.st
```iecst
(** 2018-12-07 **)
ACTION Act_RstErr:

	IF p_udiRstErr <> udiRstErrOld THEN
		bRstErr			:= TRUE;
		udiRstErrOld	:= p_udiRstErr;
	ELSE
		bRstErr			:= FALSE;
	END_IF

END_ACTION
```
